// _Internal/GroupController/Interfaces/I_ContainXtsMoverGroupController
INTERFACE I_ContainXtsMoverGroupController EXTENDS I_Base

PROPERTY XtsMoverGroupController : I_XtsMoverGroupController
SET
END_SET
END_PROPERTY

END_INTERFACE

// _Internal/GroupController/Interfaces/I_XtsMoverGroupController
INTERFACE I_XtsMoverGroupController EXTENDS I_Base, I_TaskResult, I_Resettable, I_Enablable

{attribute 'monitoring' := 'call'}
PROPERTY AxesGroup : REFERENCE TO AXES_GROUP_REF
SET
END_SET
END_PROPERTY

{attribute 'monitoring':='call'}
PROPERTY GroupStatus : E_MoverGroupState
GET
END_GET
END_PROPERTY

END_INTERFACE

// _Internal/XtsSystem/Tasks/Interfaces/I_XtsMoverIdentificationTask
INTERFACE I_XtsMoverIdentificationTask EXTENDS I_XtsTask, I_Cyclic, I_XtsExecutableTask

END_INTERFACE

// _Internal/Mover/Parameters/Interfaces/I_CollisionAvoidanceGroupable
INTERFACE I_CollisionAvoidanceGroupable EXTENDS I_Base

PROPERTY AxesGroup : REFERENCE TO AXES_GROUP_REF
GET
END_GET
SET
END_SET
END_PROPERTY

{attribute 'monitoring':='call'}
PROPERTY IdentInGroup : UDINT
GET
END_GET
SET
END_SET
END_PROPERTY

END_INTERFACE

// XtsMover/XtsMover
{attribute 'no_explicit_call' := 'This FB is a CLASS and must be accessed using methods or properties'}
FUNCTION_BLOCK XtsMover EXTENDS CyclicComponent IMPLEMENTS I_XtsMover
VAR
	_Axis				  : AXIS_REF;
	_MoverTaskCollection : XtsMoverTaskCollection<15>(THIS^);
	{attribute 'hide'}
	_VirtualMover : BOOL;
	{attribute 'hide'}
	_ManualGroupControl : BOOL;
	{attribute 'hide'}
	_MoverId : UDINT;
	{attribute 'hide'}
	_Parameters	 : XtsParameterSet;
	_CurrentTask : I_XtsMoverTaskResult := NullObjects.XtsMoverTaskResult;
	_Tasks		 : _MoverTasks;
	{attribute 'hide'}
	_MoverData : I_XtsMoverData := NullObjects.XtsMoverData;
	{attribute 'hide'}
	_oldPosition : LREAL;
	{attribute 'hide'}
	_currentPosition : LREAL;
	{attribute 'hide'}
	_TrackCollection : I_XtsTrackCollection;
	{attribute 'hide'}
	_Initialized : BOOL;
	{attribute 'hide'}
	_LocalLogger : XtsLocalLogger;
	{attribute 'hide'}
	_Logger : XtsTracePublisher;

	//
	{attribute 'hide'}
	_MoverUtility : I_TcIoXtsXpuMover;
	_Positionable : PositionableBehavior(THIS^);
	{attribute 'hide'}
	_MoverStatus : XtsMoverStatus(THIS^);
END_VAR

METHOD CyclicLogic
_MoverTaskCollection.CyclicLogic();

Axis.ReadStatus();
_oldPosition := Position;
_Positionable.CyclicLogic();
END_METHOD

PROPERTY MoverTasks : I_XtsMoverTaskCollection
GET
MoverTasks := _MoverTaskCollection;
END_GET
END_PROPERTY

PROPERTY MoverUtility : I_TcIoXtsXpuMover
GET
MoverUtility := _MoverUtility;
END_GET
SET
_MoverUtility := MoverUtility;
_Positionable.MoverUtility := _MoverUtility;
END_SET
END_PROPERTY

METHOD RefreshMoverId
VAR_INPUT
	Xpu : I_TcIoXtsProcessingUnit;
END_VAR

VAR
	MoverCount : UDINT;
	i		   : UDINT;
END_VAR
IF _VirtualMover OR _MoverUtility = 0 THEN
	RETURN;
END_IF

IF Xpu = 0 THEN
	_Logger.LogMessage(Key		 := 'RefreshMoverId',
					   Value	 := 'Invalid Xpu interface provided',
					   MessageId := E_XtsLogMessage.MoverRefreshMoverIdInvalidXpu,
					   Severity	 := 3);
END_IF

FOR i := 1 TO Xpu.P_MoverCount DO
	IF _Axis.DriveAddress.TcAxisObjectId = Xpu.MoverTcIo(UDINT_TO_UINT(i)).GetAxisObjectId() THEN
		_MoverId := i;
		RETURN;
	END_IF
END_FOR

_MoverId := 0;
_Logger.LogMessage(Key		 := 'RefreshMoverId',
				   Value	 := 'AxisId not found on XPU.',
				   MessageId := E_XtsLogMessage.MoverRefreshMoverIdNoAxisObjectFound,
				   Severity	 := 1);
END_METHOD

METHOD RegisterWithParent
VAR_INPUT
	Parent	: Core.I_ContainComponents;
END_VAR
Parent.RegisterInitialize(THIS^);
SUPER^.RegisterWithParent(Parent);
END_METHOD

//Command Mover to Activate to track
METHOD ActivateTrack : I_XtsMoverTaskResult
VAR_INPUT
	TrackId : UDINT; //Track to Activate to
END_VAR

VAR
	_TrackId   : I_TakesTrackId;
	Track	   : I_XtsTrack;
END_VAR
__QUERYINTERFACE(_Tasks.ActivateTrack, _TrackId);
ActivateTrack := _Tasks.ActivateTrack;
IF _TrackId <> 0 THEN
	_TrackId.TrackId := TrackId;
END_IF

Track						  := _TrackCollection.GetById(TrackId);
_Parameters.Track			  := Track;
_CurrentTask := ActivateTrack := _Tasks.ActivateTrack.Execute();
END_METHOD

//Add Mover to CA Group
METHOD AddToGroup : I_XtsMoverTaskResult
VAR_INPUT
	Group : REFERENCE TO AXES_GROUP_REF; //Group to Add to
	Ident : UDINT; //Ident in Group
END_VAR

VAR
	LogMessage	 : TraceMessageInfo;
	LogSource	 : TraceSourceInfo;
END_VAR
AddToGroup := _Tasks.AddToGroup;
IF NOT __ISVALIDREF(Group) THEN
	LogMessage.Severity	 := 3;
	LogMessage.Message	 := 'Invalid Parameter: AxesGroup Reference on AddToGroup Command';
	LogMessage.MessageId := E_XtsLogMessage.MoverCommandErrorInvalidParameter;
	_Logger.LogMessageInstance(LogSource, LogMessage);
	RETURN;
END_IF

_Tasks.AddToGroup.AxesGroup	   REF= Group;
_Tasks.AddToGroup.IdentInGroup := Ident;
_CurrentTask := AddToGroup	   := _Tasks.AddToGroup.Execute();
END_METHOD

METHOD Disable
VAR
	LogMessage	 : TraceMessageInfo;
	LogSource	 : TraceSourceInfo;
END_VAR
_Tasks.EnableAxis.Disable();
LogSource.SourceName := _Name;
LogMessage.Severity	 := 1;
LogMessage.Message	 := 'Mover Commanded to Disable';
LogMessage.MessageId := E_XtsLogMessage.MoverCommandedToDisable;
_Logger.LogMessageInstance(LogSource, LogMessage);
END_METHOD

METHOD Enable
VAR
	LogMessage	 :TraceMessageInfo;
	LogSource	 :TraceSourceInfo;
END_VAR
_Tasks.EnableAxis.Enable();
LogSource.SourceName := _Name;
LogMessage.Severity	 := 1;
LogMessage.Message	 := 'Mover Commanded to Enable';
LogMessage.MessageId := E_XtsLogMessage.MoverCommandedToEnable;
_Logger.LogMessageInstance(LogSource, LogMessage);
END_METHOD

//Command Mover to Halt
METHOD Halt : I_XtsMoverTaskResult
VAR_INPUT
	Deceleration : LREAL; //Rate to Decelerate
	Gap			 : LREAL; //Gap to maintain to other movers
END_VAR
Halt					 := _Tasks.HaltMover;
_Parameters.Deceleration := Deceleration;
_Parameters.Gap			 := Gap;
_CurrentTask := Halt	 := _Tasks.HaltMover.Execute();
END_METHOD

//Command Mover to MoveToPosition
METHOD MoveToPosition : I_XtsMoverTaskResult
VAR_INPUT
	Position  : LREAL; //Position to move to
	Direction : Tc3_Mc3Definitions.MC_DIRECTION := Tc3_Mc3Definitions.MC_DIRECTION.mcDirectionPositive; //Direction to move
END_VAR
_Parameters.Position		   := Position;
_Parameters.Direction		   := Direction;
_CurrentTask := MoveToPosition := _Tasks.MoveToPosition.Execute();
END_METHOD

//Command Mover to Move to a Station
METHOD MoveToStation : I_XtsMoverTaskResult
VAR_INPUT
	Station : I_XtsStation; //Station to move to
END_VAR

VAR
	LogMessage	 : TraceMessageInfo;
	LogSource	 : TraceSourceInfo;
END_VAR
IF Station = 0 THEN
    LogMessage.Severity := 3;
    LogMessage.Message := 'Invalid Parameter: Station on MoveToStation Command';
    LogMessage.MessageId := E_XtsLogMessage.MoverCommandErrorInvalidParameter;
    _Logger.LogMessageInstance(LogSource, LogMessage);
    MoveToStation := NullObjects.XtsMoverTaskResult;
    RETURN;
END_IF

_Tasks.MoveToStation.Station := Station;
_CurrentTask := _Tasks.MoveToStation.Execute();
MoveToStation := _CurrentTask;
END_METHOD

//Command a Mover to Move At Velocity endlessly
METHOD MoveVelocity : I_XtsMoverTaskResult
VAR_INPUT
	Velocity  : LREAL;																					//Velocity to move at
	Direction : Tc3_Mc3Definitions.MC_DIRECTION := Tc3_Mc3Definitions.MC_DIRECTION.mcDirectionPositive; //Direction to move
END_VAR
MoveVelocity				 := _Tasks.MoveVelocity;
_Parameters.Velocity		 := Velocity;
_Parameters.Direction		 := Direction;
_CurrentTask := MoveVelocity := _Tasks.MoveVelocity.Execute();
END_METHOD

//Command Mover to remove from CA Group
METHOD RemoveFromGroup : I_XtsMoverTaskResult
VAR_INPUT
	Group : REFERENCE TO AXES_GROUP_REF; //Group to Remvoe Mover From
	Ident : UDINT;						 //Ident of Mover in Group
END_VAR

VAR
	LogMessage : TraceMessageInfo;
	LogSource  : TraceSourceInfo;
END_VAR
RemoveFromGroup := _Tasks.RemoveFromGroup;
IF NOT __ISVALIDREF(Group) THEN
	LogMessage.Severity	 := 3;
	LogMessage.Message	 := 'Invalid Parameter: AxesGroup Reference on RemoveFromGroup Command';
	LogMessage.MessageId := E_XtsLogMessage.MoverCommandErrorInvalidParameter;
	_Logger.LogMessageInstance(LogSource, LogMessage);
	RETURN;
END_IF

_Tasks.RemoveFromGroup.AxesGroup	REF= Group;
_Tasks.RemoveFromGroup.IdentInGroup := Ident;
_CurrentTask := RemoveFromGroup		:= _Tasks.RemoveFromGroup.Execute();
END_METHOD

METHOD Reset 
VAR
	LogMessage	 : TraceMessageInfo;
	LogSource	 : TraceSourceInfo;
END_VAR
_MoverTaskCollection.Reset();
_CurrentTask := _Tasks.ResetAxis.Execute();
END_METHOD

//Command Mover to Synchronize to an Axis
METHOD SyncToAxis : I_XtsMoverTaskResult
VAR_INPUT
	Master			   : REFERENCE TO AXIS_REF; //Axis to synchronize to
	MasterSyncPosition : LREAL;					//Master synchronize position			
	SlaveSyncPosition  : LREAL;					//Slave synchronize position
END_VAR

VAR
	LogMessage : TraceMessageInfo;
	LogSource  : TraceSourceInfo;
END_VAR
IF NOT __ISVALIDREF(Master) THEN
	LogMessage.Severity	 := 3;
	LogMessage.Message	 := 'Invalid Parameter: Master reference on SyncToAxis command';
	LogMessage.MessageId := E_XtsLogMessage.MoverCommandErrorInvalidParameter;
	_Logger.LogMessageInstance(LogSource, LogMessage);
	RETURN;
END_IF

_Parameters.SyncAxis.MasterAxis			REF= Master;
_Parameters.SyncAxis.MasterSyncPosition := MasterSyncPosition;
_Parameters.SyncAxis.SlaveSyncPosition	:= SlaveSyncPosition;
_CurrentTask := SyncToAxis				:= _Tasks.SyncToAxis.Execute();
END_METHOD

//Command Mover to Synchronize to another Mover
METHOD SyncToMover : I_XtsMoverTaskResult
VAR_INPUT
	Master	 : I_XtsMover; //Mover to synchronize to
	Distance : LREAL;	   //Distance between movers
END_VAR

VAR
	LogMessage : TraceMessageInfo;
	LogSource  : TraceSourceInfo;
END_VAR
IF Master = 0 THEN
	LogMessage.Severity	 := 3;
	LogMessage.Message	 := 'Invalid Parameter: Master on SyncToMover Command';
	LogMessage.MessageId := E_XtsLogMessage.MoverCommandErrorInvalidParameter;
	_Logger.LogMessageInstance(LogSource, LogMessage);
	RETURN;
END_IF

_Parameters.SyncAxis.MasterAxis			REF= Master.Axis;
_Parameters.SyncAxis.MasterSyncPosition := Master.Axis.NcToPlc.SetPos;
IF _Axis.NcToPlc.SetPos <= Master.Axis.NcToPlc.SetPos THEN
	IF Distance > 0 THEN		// ... And the Gap is Positive
		_Parameters.SyncAxis.SlaveSyncPosition		:= Master.Axis.NcToPlc.SetPos - Distance;		
	ELSE				// ... And the Gap is Negative
		_Parameters.SyncAxis.SlaveSyncPosition		:= Master.Axis.NcToPlc.SetPos - Status.CurrentTrack.Length - Distance;
	END_IF

// If the slave setpos is greater than the master...
ELSE
	IF Distance > 0 THEN		// ... And the Gap is Positive
		_Parameters.SyncAxis.SlaveSyncPosition		:= Master.Axis.NcToPlc.SetPos - Status.CurrentTrack.Length - Distance;
	ELSE				// ... And the Gap is Negative
		_Parameters.SyncAxis.SlaveSyncPosition		:= Master.Axis.NcToPlc.SetPos - Distance;		
	END_IF
END_IF
_CurrentTask := SyncToMover				:= _Tasks.SyncToAxis.Execute();
LogSource.SourceName					:= _Name;
END_METHOD

//FB_Init is always available implicitly and it is used primarily for initialization.

//The return value is not evaluated. For a specific influence, you can also declare the

//methods explicitly and provide additional code there with the standard initialization

//code. You can evaluate the return value.
METHOD FB_Init : BOOL
VAR_INPUT
	bInitRetains : BOOL; // TRUE: the retain variables are initialized (reset warm / reset cold)
	bInCopyCode	 : BOOL; // TRUE: the instance will be copied to the copy code afterward (online change)
	Name		 : T_MaxString;
	MoverData	 : I_XtsMoverData;		   //Optional MoverData assignment
	System		 : I_ContainXtsMovers; //Optional Self Registration with an Xts System
END_VAR
_MoverTaskCollection.AddTask(_Tasks.EnableAxis);
_MoverTaskCollection.AddTask(_Tasks.ResetAxis);
_MoverTaskCollection.AddTask(_Tasks.MoveToPosition);
_MoverTaskCollection.AddTask(_Tasks.MoveToStation);
_MoverTaskCollection.AddTask(_Tasks.MoveVelocity);
_MoverTaskCollection.AddTask(_Tasks.HaltMover);
_MoverTaskCollection.AddTask(_Tasks.AddToGroup);
_MoverTaskCollection.AddTask(_Tasks.RemoveFromGroup);
_MoverTaskCollection.AddTask(_Tasks.ActivateTrack);
_MoverTaskCollection.AddTask(_Tasks.SyncToAxis);
_Logger.Subscribe(_LocalLogger);
IF XtsCoreParameters.TcEventLoggerEnabled THEN
	_Logger.Subscribe(XtsTrace.EventLogger);
END_IF

IF MoverData <> 0 THEN
	_MoverData := MoverData;
END_IF

IF System <> 0 THEN
	System.Movers.AddItem(THIS^);
	RegisterWithParent(System);
END_IF
END_METHOD

METHOD Initialize
VAR
	CurrentTrackOtcid : OTCID;
END_VAR
IF _TrackCollection = 0 THEN
	RETURN;
END_IF


IF _MoverUtility = 0 OR _VirtualMover THEN
	_Initialized := TRUE;	
	RETURN;
END_IF

CurrentTrackOtcid := _MoverUtility.GetActiveTrackObjectId();
_TrackCollection.ResetIterator();
WHILE _TrackCollection.MoveToNext DO
	IF _TrackCollection.Current.Otcid = CurrentTrackOtcid THEN
		_MoverStatus.CurrentTrack := _TrackCollection.Current;
		EXIT;
	END_IF
END_WHILE

_Initialized := TRUE;
END_METHOD

{attribute 'monitoring' := 'call'}
PROPERTY Initialized : BOOL
GET
Initialized := _Initialized;
END_GET
SET
_Initialized := Initialized;
END_SET
END_PROPERTY

PROPERTY Axis : REFERENCE TO Tc2_MC2.AXIS_REF
GET
Axis REF= _Axis;
END_GET
END_PROPERTY

{attribute 'monitoring' := 'call'}
PROPERTY InhibitFeedBackward : BOOL
GET
InhibitFeedBackward := _Tasks.EnableAxis.InhibitFeedBackward;
END_GET
SET
_Tasks.EnableAxis.InhibitFeedBackward := InhibitFeedBackward;
END_SET
END_PROPERTY

{attribute 'monitoring' := 'call'}
PROPERTY InhibitFeedForward : BOOL
GET
InhibitFeedForward := _Tasks.EnableAxis.InhibitFeedForward;
END_GET
SET
_Tasks.EnableAxis.InhibitFeedForward := InhibitFeedForward;
END_SET
END_PROPERTY

{attribute 'monitoring':='call'}
PROPERTY InPosition : BOOL
GET
VAR
	difference : LREAL;
END_VAR
difference := ABS(Position - _Parameters.Position);
InPosition := MIN(difference, _Parameters.Track.Length - difference) < 1.0 AND (NOT _Tasks.MoveToPosition.Busy OR NOT _Tasks.MoveToStation.Busy);
END_GET
END_PROPERTY

{attribute 'monitoring':='call'}
PROPERTY InVelocity : BOOL
GET
InVelocity := ABS(_Axis.NcToPlc.ActVelo -  _Axis.NcToPlc.SetVelo) < 10.0 AND _Axis.NcToPlc.SetVelo <> 0;
END_GET
END_PROPERTY

PROPERTY LastCyclePosition : LREAL
GET
LastCyclePosition := _oldPosition;
END_GET
END_PROPERTY

{attribute 'monitoring':='call'}
PROPERTY ManualGroupControl : BOOL
GET
ManualGroupControl := _ManualGroupControl;
END_GET
SET
_ManualGroupControl := ManualGroupControl;
END_SET
END_PROPERTY

{attribute 'monitoring':='call'}
PROPERTY MoverData : I_XtsMoverData
GET
MoverData := _MoverData;
END_GET
SET
_MoverData := MoverData;
END_SET
END_PROPERTY

{attribute 'monitoring':='call'}
PROPERTY MoverId : UDINT
GET
MoverId := _MoverId;
END_GET
END_PROPERTY

{attribute 'monitoring' := 'call'}
PROPERTY Override : LREAL
SET
_Tasks.EnableAxis.Override := Override;
END_SET
END_PROPERTY

{attribute 'monitoring':='call'}
PROPERTY Parameters : I_XtsParameterSet
GET
Parameters := _Parameters;
END_GET
SET
END_SET
END_PROPERTY

{attribute 'monitoring':='call'}
PROPERTY Position : LREAL
GET
VAR
	tmp : LREAL;
END_VAR
Position := _Positionable.Position;
END_GET
END_PROPERTY

{attribute 'hide'}
PROPERTY Tracks : I_XtsTrackCollection
GET
Tracks := _TrackCollection;
END_GET
SET
_TrackCollection := Tracks;
//Reset the Activate Task axis assignment to refresh track collection assignment
_Tasks.ActivateTrack.Axis := THIS^;
END_SET
END_PROPERTY

{attribute 'monitoring':='call'}
PROPERTY VirtualMover : BOOL
GET
VirtualMover := _VirtualMover;
END_GET
SET
_VirtualMover := VirtualMover;
END_SET
END_PROPERTY

{attribute 'monitoring':='call'}
PROPERTY Busy : BOOL
GET
Busy := _MoverTaskCollection.Busy;
END_GET
END_PROPERTY

{attribute 'monitoring':='call'}
//Last Commanded Task to Mover
PROPERTY CurrentTask : I_XtsMoverTaskResult
GET
CurrentTask := _CurrentTask;
END_GET
END_PROPERTY

{attribute 'monitoring' := 'call'}
PROPERTY Enabled : BOOL
GET
Enabled := _Tasks.EnableAxis.Enabled;
END_GET
END_PROPERTY

{attribute 'monitoring':='call'}
PROPERTY Error : BOOL
GET
Error := _MoverTaskCollection.Error;
END_GET
END_PROPERTY

{attribute 'monitoring':='call'}
PROPERTY ErrorId : UDINT
GET
IF _Axis.Status.ErrorID <> 0 THEN
	ErrorId := _Axis.Status.ErrorID;
	RETURN;
END_IF

ErrorId := _MoverTaskCollection.ErrorId;
END_GET
END_PROPERTY

{attribute 'monitoring':='call'}
PROPERTY Status : I_XtsMoverStatus
GET
Status := _MoverStatus;
END_GET
END_PROPERTY

{attribute 'monitoring':='call'}
PROPERTY CommandLog : I_XtsLocalLog
GET
CommandLog := _LocalLogger;
END_GET
END_PROPERTY

PROPERTY TracePublisher : I_XtsTracePublisher
GET
TracePublisher := _Logger;
END_GET
END_PROPERTY

METHOD AcceptMoverVisitor
VAR_INPUT
	MoverVisitor : I_XtsMoverVisitor;
END_VAR
MoverVisitor.VisitMover(THIS^);
END_METHOD

END_FUNCTION_BLOCK

// _Internal/Mover/MoverTaskBase/XtsMoverTaskCollection
{attribute 'no_explicit_call' := 'This FB is a CLASS and must be accessed using methods or properties'}
FUNCTION_BLOCK XtsMoverTaskCollection
VAR_GENERIC CONSTANT
	MaxCount : UDINT := 10;
END_VAR IMPLEMENTS I_XtsMoverTaskCollection, I_Cyclic
VAR
	MotionTasks : ARRAY[0..MaxCount - 1] OF I_XtsMoverTask;
	_TaskCount	: UDINT;
	Axis		: I_AxisRef;
	_ErrorId	: UDINT;
	_Busy		: BOOL;
	_Error		: BOOL;
	_ErrorTask	: T_MaxString;
	{attribute 'hide'}
	_Logger : I_XtsLogger;
	{attribute 'hide'}
	LogSource : TraceSourceInfo;
	{attribute 'hide'}
	LogMessage : TraceMessageInfo;
END_VAR

PROPERTY Busy : BOOL
GET
Busy := _Busy;
END_GET
END_PROPERTY

PROPERTY Error : BOOL
GET
Error := _Error;
END_GET
END_PROPERTY

PROPERTY ErrorId : UDINT
GET
ErrorId := _ErrorId;
END_GET
END_PROPERTY

PROPERTY ErrorTask : T_MaxString
GET
ErrorTask := _ErrorTask;
END_GET
END_PROPERTY

METHOD AddTask : BOOL
VAR_INPUT
	Task	: I_XtsMoverTask;
END_VAR
IF _TaskCount = MaxCount THEN
	AddTask := FALSE;
	RETURN;
END_IF
Task.Axis := Axis;
MotionTasks[Task.TaskId] := Task;
_TaskCount := _TaskCount + 1;
AddTask := TRUE;
END_METHOD

METHOD CyclicLogic
VAR
	i	 : UDINT;
END_VAR
_Busy := FALSE;
FOR i := 0 TO MaxCount - 1 DO
	IF MotionTasks[i] = 0 THEN
		CONTINUE;
	END_IF

	MotionTasks[i].CyclicLogic();
	IF MotionTasks[i].Busy THEN
		_Busy := TRUE;
	END_IF

	IF MotionTasks[i].Error AND NOT _Error THEN
		LogMessage.Message	 := CONCAT('Mover Task: ', CONCAT(MotionTasks[i].TaskName, CONCAT(' ErrorId: ', TO_STRING(MotionTasks[i].ErrorId))));
		LogMessage.MessageId := E_XtsLogMessage.MoverCommandGeneralTaskError;
		LogMessage.Severity	 := 3;
		_Logger.LogMessageInstance(LogSource, LogMessage);
		_Error	   := TRUE;
		_ErrorId   := MotionTasks[i].ErrorId;
		_ErrorTask := MotionTasks[i].TaskName;
	END_IF
END_FOR
END_METHOD

//FB_Init is always available implicitly and it is used primarily for initialization.

//The return value is not evaluated. For a specific influence, you can also declare the

//methods explicitly and provide additional code there with the standard initialization

//code. You can evaluate the return value.
METHOD FB_Init : BOOL
VAR_INPUT
	bInitRetains : BOOL; // TRUE: the retain variables are initialized (reset warm / reset cold)
	bInCopyCode	 : BOOL; // TRUE: the instance will be copied to the copy code afterward (online change)
	Axis		 : I_AxisRef;
END_VAR
VAR
	Mover : I_XtsMover;
END_VAR
THIS^.Axis			 := Axis;
LogSource.SourceName := 'Task Collection';
__QUERYINTERFACE(Axis, Mover);
__QUERYINTERFACE(Mover.TracePublisher, _Logger);
END_METHOD

METHOD GetTaskById : I_XtsMoverTask
VAR_INPUT
	TaskId : MoverTaskID;
END_VAR
GetTaskById := MotionTasks[TaskId];
END_METHOD

METHOD GetTaskByName : I_XtsMoverTask
VAR_INPUT
	Name : T_MaxString;
END_VAR

VAR
	i	 : UDINT;
END_VAR
GetTaskByName := NullObjects.XtsMoverTask;
FOR i:=0 TO _TaskCount - 1 DO
	IF MotionTasks[i].TaskName = Name THEN
		GetTaskByName := MotionTasks[i];
		RETURN;
	END_IF
END_FOR
END_METHOD

METHOD RemoveTaskById : BOOL
VAR_INPUT
	TaskId : MoverTaskId;
END_VAR
IF MotionTasks[TaskId] = 0 THEN
	RETURN;
END_IF

MotionTasks[TaskId] := 0;
_TaskCount			:= _TaskCount - 1;
RemoveTaskById		:= TRUE;
END_METHOD

METHOD RemoveTaskByInstance : BOOL
VAR_INPUT
	Task : I_XtsMoverTask;
END_VAR
IF MotionTasks[Task.TaskId] = 0 THEN
	RETURN;
END_IF

MotionTasks[Task.TaskId] := 0;
_TaskCount				 := _TaskCount - 1;
RemoveTaskByInstance	 := TRUE;
END_METHOD

METHOD Reset
VAR_INPUT
END_VAR
VAR
	i : UDINT;
END_VAR
_Error	   := FALSE;
_ErrorId   := 0;
_ErrorTask := '';
FOR i := 0 TO MaxCount - 1 DO
	IF MotionTasks[i] = 0 THEN
		CONTINUE;
	END_IF
	MotionTasks[i].Reset();
END_FOR
END_METHOD

END_FUNCTION_BLOCK

// _Internal/Mover/Tasks/_MoverTasks
{attribute 'no_explicit_call' := 'This FB is a CLASS and must be accessed using methods or properties'}
FUNCTION_BLOCK _MoverTasks
VAR
	_DefaultTask	 : _DefaultMoverTasks;
	_MoveToPosition	 : I_XtsMoverTask		:= _DefaultTask.MoveToPositionCA;
	_MoveVelocity	 : I_XtsMoverTask		:= _DefaultTask.MoveVelocity;
	_HaltMoverCA	 : I_XtsMoverTask		:= _DefaultTask.HaltMoverCA;
	_AddToGroup		 : I_AxesGroupTask		:= _DefaultTask.AddToGroup;
	_RemoveFromGroup : I_AxesGroupTask		:= _DefaultTask.RemoveFromGroup;
	_MoveToStation	 : I_MoveToStationTask	:= _DefaultTask.MoveToStation;
	_ActivateTrack	 : I_XtsMoverTask		:= _DefaultTask.ActivateTrack;
	_EnableAxis		 : I_EnableXtsMoverTask := _DefaultTask.EnableAxis;
	_ResetAxis		 : I_XtsMoverTask		:= _DefaultTask.ResetAxis;
	_SyncToAxis		 : I_XtsMoverTask		:= _DefaultTask.SyncToAxis;
END_VAR

PROPERTY ActivateTrack : I_XtsMoverTask
GET
ActivateTrack := _ActivateTrack;
END_GET
SET
_ActivateTrack := ActivateTrack;
END_SET
END_PROPERTY

PROPERTY AddToGroup : I_AxesGroupTask
GET
AddToGroup := _AddToGroup;
END_GET
SET
_AddToGroup := AddToGroup;
END_SET
END_PROPERTY

PROPERTY EnableAxis : I_EnableXtsMoverTask
GET
EnableAxis := _EnableAxis;
END_GET
SET
_EnableAxis := EnableAxis;
END_SET
END_PROPERTY

PROPERTY HaltMover : I_XtsMoverTask
GET
HaltMover := _HaltMoverCA;
END_GET
SET
_HaltMoverCA := HaltMover;
END_SET
END_PROPERTY

PROPERTY MoveToPosition : I_XtsMoverTask
GET
MoveToPosition := _MoveToPosition;
END_GET
SET
_MoveToPosition := MoveToPosition;
END_SET
END_PROPERTY

PROPERTY MoveToStation : I_MoveToStationTask
GET
MoveToStation := _MoveToStation;
END_GET
SET
_MoveToStation := MoveToStation;
END_SET
END_PROPERTY

PROPERTY MoveVelocity : I_XtsMoverTask
GET
MoveVelocity := _MoveVelocity;
END_GET
SET
_MoveVelocity := MoveVelocity;
END_SET
END_PROPERTY

PROPERTY RemoveFromGroup : I_AxesGroupTask
GET
RemoveFromGroup := _RemoveFromGroup;
END_GET
SET
_RemoveFromGroup := RemoveFromGroup;
END_SET
END_PROPERTY

PROPERTY ResetAxis : I_XtsMoverTask
GET
ResetAxis := _ResetAxis;
END_GET
SET
_ResetAxis := ResetAxis;
END_SET
END_PROPERTY

METHOD ResetToDefault
VAR_INPUT
END_VAR
_MoveToPosition	 := _DefaultTask.MoveToPositionCA;
_MoveVelocity	 := _DefaultTask.MoveVelocity;
_HaltMoverCA	 := _DefaultTask.HaltMoverCA;
_AddToGroup		 := _DefaultTask.AddToGroup;
_RemoveFromGroup := _DefaultTask.RemoveFromGroup;
_MoveToStation	 := _DefaultTask.MoveToStation;
_ActivateTrack	 := _DefaultTask.ActivateTrack;
_EnableAxis		 := _DefaultTask.EnableAxis;
_ResetAxis		 := _DefaultTask.ResetAxis;
_SyncToAxis		 := _DefaultTask.SyncToAxis;
END_METHOD

PROPERTY SyncToAxis : I_XtsMoverTask
GET
SyncToAxis := _SyncToAxis;
END_GET
SET
_SyncToAxis := SyncToAxis;
END_SET
END_PROPERTY

END_FUNCTION_BLOCK

// _Internal/Mover/Tasks/_DefaultMoverTasks
{attribute 'no_explicit_call' := 'This FB is a CLASS and must be accessed using methods or properties'}
FUNCTION_BLOCK _DefaultMoverTasks
VAR
	NullMotionTask	 : NullXtsMoverTask;
	EnableAxis		 : EnableAxisTask;
	AddToGroup		 : AddToGroupTask;
	RemoveFromGroup	 : RemoveFromGroupTask;
	HaltMoverCA		 : HaltMoverCATask;
	MoveToPositionCA : MoveToPositionCATask;
	MoveVelocity	 : MoveVelocityTask;
	MoveToStation	 : MoveToStationTask;
	ActivateTrack	 : ActivateTrackTask;
	ResetAxis		 : ResetAxisTask;
	SyncToAxis		 : SyncToAxisTask;
END_VAR

END_FUNCTION_BLOCK

// _Internal/NullObjects/NullXtsMoverTask
{attribute 'no_explicit_call' := 'This FB is a CLASS and must be accessed using methods or properties'}
{attribute 'conditionalshow'}
{warning disable C0094}
{warning disable C0568}
FUNCTION_BLOCK NullXtsMoverTask EXTENDS XtsMoverTaskResult IMPLEMENTS I_XtsMoverTask, I_NullObject
VAR
END_VAR

PROPERTY Axis : I_AxisRef
GET
END_GET
SET
END_SET
END_PROPERTY

METHOD CyclicLogic
END_METHOD

METHOD Execute : I_XtsMoverTaskResult
Execute := NullObjects.XtsMoverTaskResult;
END_METHOD

METHOD Reset
END_METHOD

PROPERTY TaskId : MoverTaskId
GET
END_GET
END_PROPERTY

{attribute 'monitoring':='call'}
PROPERTY TaskName : STRING
GET
TaskName := 'No task active';
END_GET
END_PROPERTY

END_FUNCTION_BLOCK

// _Internal/Mover/Tasks/EnableAxisTask
{attribute 'no_explicit_call' := 'This FB is a CLASS and must be accessed using methods or properties'}
FUNCTION_BLOCK EnableAxisTask EXTENDS XtsMoverTaskResult IMPLEMENTS I_EnableXtsMoverTask
VAR
	_Axis			   : I_AxisRef;
	_DefaultAxisEnable : PowerAxis;
	EnableAxisFb	   : I_Power := _DefaultAxisEnable;
	{attribute 'hide'}
	_InhibitFeedForward : BOOL;
	{attribute 'hide'}
	_InhibitFeedBackward : BOOL;
END_VAR

PROPERTY Axis : I_AxisRef
GET
Axis := _Axis;
END_GET
SET
_Axis := Axis;
END_SET
END_PROPERTY

METHOD CyclicLogic
EnableAxisFb.Enable_Positive := NOT _InhibitFeedForward;
EnableAxisFb.Enable_Negative := NOT _InhibitFeedBackward;
_DefaultAxisEnable(Axis := _Axis.Axis);
_Error	 := EnableAxisFb.Error;
_Busy	 := EnableAxisFb.Busy AND NOT EnableAxisFb.Status;
_ErrorId := EnableAxisFb.ErrorId;
END_METHOD

METHOD Disable
EnableAxisFb.Enable := FALSE;
END_METHOD

{attribute 'monitoring' := 'call'}
PROPERTY Disabled : BOOL
GET
Disabled := EnableAxisFb.Status = FALSE;
END_GET
END_PROPERTY

METHOD Enable
EnableAxisFb.Enable := TRUE;
END_METHOD

{attribute 'monitoring' := 'call'}
PROPERTY Enabled : BOOL
GET
Enabled := EnableAxisFb.Status;
END_GET
END_PROPERTY

METHOD Execute : I_XtsMoverTaskResult
Execute := THIS^;
END_METHOD

//FB_Init is always available implicitly and it is used primarily for initialization.

//The return value is not evaluated. For a specific influence, you can also declare the

//methods explicitly and provide additional code there with the standard initialization

//code. You can evaluate the return value.
METHOD FB_Init : BOOL
VAR_INPUT
	bInitRetains : BOOL; // TRUE: the retain variables are initialized (reset warm / reset cold)
	bInCopyCode	 : BOOL; // TRUE: the instance will be copied to the copy code afterward (online change)
END_VAR
_TaskName := 'Enable Axis';
_TaskId	  := MoverTaskId.ENABLE;
END_METHOD

{attribute 'monitoring' := 'call'}
PROPERTY InhibitFeedBackward : BOOL
GET
InhibitFeedBackward := _InhibitFeedBackward;
END_GET
SET
_InhibitFeedBackward := InhibitFeedBackward;
END_SET
END_PROPERTY

{attribute 'monitoring' := 'call'}
PROPERTY InhibitFeedForward : BOOL
GET
InhibitFeedForward := _InhibitFeedForward;
END_GET
SET
_InhibitFeedForward := InhibitFeedForward;
END_SET
END_PROPERTY

{attribute 'monitoring' := 'call'}
PROPERTY Override : LREAL
SET
EnableAxisFb.Override := Override;
END_SET
END_PROPERTY

METHOD Reset
_Error				 := FALSE;
_ErrorID			 := 0;
_Busy				 := FALSE;
ExecuteWatchdog		 := 0;
_CommandExecuted	 := FALSE;
END_METHOD

END_FUNCTION_BLOCK

// _Internal/Mover/Tasks/Interfaces/I_EnableXtsMoverTask
INTERFACE I_EnableXtsMoverTask EXTENDS I_XtsMoverTask, I_Cyclic

METHOD Disable
END_METHOD

{attribute 'monitoring' := 'call'}
PROPERTY Disabled : BOOL
GET
END_GET
END_PROPERTY

METHOD Enable
END_METHOD

{attribute 'monitoring' := 'call'}
PROPERTY Enabled : BOOL
GET
END_GET
END_PROPERTY

{attribute 'monitoring' := 'call'}
PROPERTY InhibitFeedBackward : BOOL
GET
END_GET
SET
END_SET
END_PROPERTY

{attribute 'monitoring' := 'call'}
PROPERTY InhibitFeedForward : BOOL
GET
END_GET
SET
END_SET
END_PROPERTY

{attribute 'monitoring' := 'call'}
PROPERTY Override : LREAL
SET
END_SET
END_PROPERTY

END_INTERFACE

// _Internal/Mover/Tasks/Wrappers/PowerAxis
FUNCTION_BLOCK PowerAxis IMPLEMENTS I_Power
VAR
	_mcPower : MC_Power;
END_VAR

VAR_IN_OUT
	Axis : Tc2_Mc2.AXIS_REF;
END_VAR

_mcPower(Axis := Axis);

{attribute 'monitoring':='call'}
PROPERTY BufferMode : MC_BufferMode
GET
BufferMode := _mcPower.BufferMode;
END_GET
SET
_mcPower.BufferMode := BufferMode;
END_SET
END_PROPERTY

{attribute 'monitoring':='call'}
PROPERTY Enable : BOOL
GET
Enable := _mcPower.Enable;
END_GET
SET
_mcPower.Enable := Enable;
END_SET
END_PROPERTY

{attribute 'monitoring':='call'}
PROPERTY Enable_Negative : BOOL;
GET
Enable_Negative := _mcPower.Enable_Negative;
END_GET
SET
_mcPower.Enable_Negative := Enable_Negative;
END_SET
END_PROPERTY

{attribute 'monitoring':='call'}
PROPERTY Enable_Positive : BOOL
GET
Enable_Positive := _mcPower.Enable_Positive;
END_GET
SET
_mcPower.Enable_Positive := Enable_Positive;
END_SET
END_PROPERTY

PROPERTY Options : ST_PowerOptions
GET
Options := _mcPower.Options;
END_GET
SET
_mcPower.Options := Options;
END_SET
END_PROPERTY

{attribute 'monitoring':='call'}
PROPERTY Override : MC_LREAL
GET
Override := _mcPower.Override;
END_GET
SET
_mcPower.Override := Override;
END_SET
END_PROPERTY

{attribute 'monitoring':='call'}
PROPERTY Busy : BOOL
GET
Busy := _mcPower.Busy;
END_GET
END_PROPERTY

{attribute 'monitoring':='call'}
PROPERTY Error : BOOL
GET
Error := _mcPower.Error;
END_GET
END_PROPERTY

{attribute 'monitoring':='call'}
PROPERTY ErrorId : UDINT
GET
ErrorId := _mcPower.ErrorID;
END_GET
END_PROPERTY

{attribute 'monitoring':='call'}
PROPERTY Status : BOOL
GET
Status := _mcPower.Status;
END_GET
END_PROPERTY

END_FUNCTION_BLOCK

// _Internal/Mover/Tasks/Wrappers/Interfaces/I_Power
INTERFACE I_Power EXTENDS I_Base

{attribute 'monitoring':='call'}
PROPERTY BufferMode : MC_BufferMode
GET
END_GET
SET
END_SET
END_PROPERTY

{attribute 'monitoring':='call'}
PROPERTY Enable : BOOL
GET
END_GET
SET
END_SET
END_PROPERTY

{attribute 'monitoring':='call'}
PROPERTY Enable_Negative : BOOL;
GET
END_GET
SET
END_SET
END_PROPERTY

{attribute 'monitoring':='call'}
PROPERTY Enable_Positive : BOOL
GET
END_GET
SET
END_SET
END_PROPERTY

PROPERTY Options : ST_PowerOptions
GET
END_GET
SET
END_SET
END_PROPERTY

{attribute 'monitoring':='call'}
PROPERTY Override : MC_LREAL
GET
END_GET
SET
END_SET
END_PROPERTY

{attribute 'monitoring':='call'}
PROPERTY Busy : BOOL
GET
END_GET
END_PROPERTY

{attribute 'monitoring':='call'}
PROPERTY Error : BOOL
GET
END_GET
END_PROPERTY

{attribute 'monitoring':='call'}
PROPERTY ErrorId : UDINT
GET
END_GET
END_PROPERTY

{attribute 'monitoring':='call'}
PROPERTY Status : BOOL
GET
END_GET
END_PROPERTY

END_INTERFACE

// _Internal/Mover/Tasks/AddToGroupTask
{attribute 'no_explicit_call' := 'This FB is a CLASS and must be accessed using methods or properties'}
FUNCTION_BLOCK AddToGroupTask EXTENDS XtsMoverTaskResult IMPLEMENTS I_AxesGroupTask
VAR
	_Axis				   : I_AxisRef;
	_MoverStatus		   : I_XtsMoverStatus;
	_DefaultAddAxisToGroup : AddAxisToGroup;
	AddToGroupFb		   : I_AxisOnGroup := _DefaultAddAxisToGroup;
	_AxesGroup			   : REFERENCE TO AXES_GROUP_REF;
	_Ident				   : UDINT;
	Executed			   : BOOL;
END_VAR

PROPERTY AxesGroup : REFERENCE TO AXES_GROUP_REF
GET
AxesGroup REF= _AxesGroup;
END_GET
SET
_AxesGroup REF= AxesGroup;
END_SET
END_PROPERTY

PROPERTY Axis : I_AxisRef
GET
Axis := _Axis;
END_GET
SET
VAR
	Mover : I_XtsMover;
END_VAR
_Axis := Axis;
__QUERYINTERFACE(_Axis, Mover);
__QUERYINTERFACE(Mover.TracePublisher, _Logger);
_MoverStatus := Mover.Status;
END_SET
END_PROPERTY

METHOD CyclicLogic
SUPER^.CyclicLogic(); //Watchdog handling
_DefaultAddAxisToGroup(Axis := _Axis.Axis, AxesGroup := _AxesGroup);
AddToGroupFb.Execute := FALSE;
_Busy				 := AddToGroupFb.Busy;
IF _Busy THEN
	RETURN;
END_IF

(*Latch signals if they are set by the FB instance itself.
Only reset them in the event of an Task.Execute() call*)
IF Executed THEN
	Executed				  := FALSE;
	_MoverStatus.IdentInGroup := _Ident;
END_IF

_Error := AddToGroupFb.Error OR _Error;
IF AddToGroupFb.ErrorId <> 0 THEN
	_ErrorId := AddToGroupFb.ErrorId;
END_IF
END_METHOD

METHOD Execute : I_XtsMoverTaskResult
Execute			:= THIS^;
ExecuteWatchdog := ExecuteWatchdog + 1;
IF NOT __ISVALIDREF(_AxesGroup) OR _Ident = 0 THEN
	//TODO: error message
	RETURN;
END_IF

IF _Busy OR _CommandExecuted THEN
	RETURN;
END_IF

_Error					  := FALSE;
_ErrorId				  := 0;
_Busy					  := TRUE;
AddToGroupFb.IdentInGroup := _Ident;
AddToGroupFb.Execute	  := TRUE;
_CommandExecuted		  := TRUE;
Executed				  := TRUE;
LogMessage.Severity		  := 1;
LogMessage.Message		  := 'Commanded to Add to Group.';
LogMessage.MessageId	  := E_XtsLogMessage.MoverCommandedToAddToGroup;
_Logger.LogMessageInstance(LogSource, LogMessage);
END_METHOD

//FB_Init is always available implicitly and it is used primarily for initialization.

//The return value is not evaluated. For a specific influence, you can also declare the

//methods explicitly and provide additional code there with the standard initialization

//code. You can evaluate the return value.
METHOD FB_Init : BOOL
VAR_INPUT
	bInitRetains : BOOL; // TRUE: the retain variables are initialized (reset warm / reset cold)
	bInCopyCode	 : BOOL; // TRUE: the instance will be copied to the copy code afterward (online change)
END_VAR
_TaskName			 := 'Add Axis To Group';
_TaskId				 := MoverTaskId.ADD_TO_GROUP;
LogSource.SourceName := _TaskName;
LogSource.SourceId	 := _TaskId;
END_METHOD

{attribute 'monitoring':='call'}
PROPERTY IdentInGroup : UDINT
GET
IdentInGroup := _Ident;
END_GET
SET
_Ident := IdentInGroup;
END_SET
END_PROPERTY

METHOD Reset
Executed			 := FALSE;
_Error				 := FALSE;
_ErrorID			 := 0;
_Busy				 := FALSE;
ExecuteWatchdog		 := 0;
_CommandExecuted	 := FALSE;
AddToGroupFb.Execute := FALSE;
END_METHOD

END_FUNCTION_BLOCK

// _Internal/Mover/Tasks/Interfaces/I_AxesGroupTask
INTERFACE I_AxesGroupTask EXTENDS I_Base, I_XtsMoverTask, I_CollisionAvoidanceGroupable

END_INTERFACE

// _Internal/Mover/Tasks/Wrappers/AddAxisToGroup
FUNCTION_BLOCK AddAxisToGroup IMPLEMENTS I_AxisOnGroup
VAR
	_AddAxisToGroup : MC_AddAxisToGroup;
	_Ident			: UDINT;
END_VAR

VAR_IN_OUT
	Axis	  : Tc2_Mc2.AXIS_REF;
	AxesGroup : Tc3_McCoordinatedMotion.AXES_GROUP_REF;
END_VAR

_AddAxisToGroup(Axis := Axis, AxesGroup := AxesGroup);

{attribute 'monitoring':='call'}
PROPERTY Execute : BOOL
GET
Execute := _AddAxisToGroup.Execute;
END_GET
SET
_AddAxisToGroup.Execute := Execute;
END_SET
END_PROPERTY

{attribute 'monitoring':='call'}
PROPERTY IdentInGroup : UDINT
GET
IdentInGroup := _Ident;
END_GET
SET
_Ident := IdentInGroup;
_AddAxisToGroup.IdentInGroup :=UDINT_TO_IDENTINGROUP(IdentInGroup);
END_SET
END_PROPERTY

{attribute 'monitoring':='call'}
PROPERTY Busy : BOOL
GET
Busy := _AddAxisToGroup.Busy;
END_GET
END_PROPERTY

{attribute 'monitoring':='call'}
PROPERTY Done : BOOL
GET
Done := _AddAxisToGroup.Done;
END_GET
END_PROPERTY

{attribute 'monitoring':='call'}
PROPERTY Error : BOOL
GET
Error := _AddAxisToGroup.Error;
END_GET
END_PROPERTY

{attribute 'monitoring':='call'}
PROPERTY ErrorId : UDINT
GET
ErrorId := _AddAxisToGroup.ErrorId;
END_GET
END_PROPERTY

END_FUNCTION_BLOCK

// _Internal/Mover/Tasks/Wrappers/Interfaces/I_AxisOnGroup
INTERFACE I_AxisOnGroup EXTENDS I_Base

{attribute 'monitoring':='call'}
PROPERTY Execute : BOOL
GET
END_GET
SET
END_SET
END_PROPERTY

{attribute 'monitoring':='call'}
PROPERTY IdentInGroup : UDINT
GET
END_GET
SET
END_SET
END_PROPERTY

{attribute 'monitoring':='call'}
PROPERTY Busy : BOOL
GET
END_GET
END_PROPERTY

{attribute 'monitoring':='call'}
PROPERTY Error : BOOL
GET
END_GET
END_PROPERTY

{attribute 'monitoring':='call'}
PROPERTY ErrorId : UDINT
GET
END_GET
END_PROPERTY

END_INTERFACE

// _Internal/Mover/Tasks/RemoveFromGroupTask
{attribute 'no_explicit_call' := 'This FB is a CLASS and must be accessed using methods or properties'}
FUNCTION_BLOCK RemoveFromGroupTask EXTENDS XtsMoverTaskResult IMPLEMENTS I_AxesGroupTask
VAR
	_Axis						: I_AxisRef;
	_MoverStatus				: I_XtsMoverStatus;
	_DefaultRemoveAxisFromGroup : RemoveAxisFromGroup;
	RemoveFromGroupFb			: I_AxisOnGroup := _DefaultRemoveAxisFromGroup;
	_AxesGroup					: REFERENCE TO AXES_GROUP_REF;
	_Ident						: UDINT;
	Executed					: BOOL;
END_VAR

PROPERTY AxesGroup : REFERENCE TO AXES_GROUP_REF
GET
AxesGroup REF= _AxesGroup;
END_GET
SET
_AxesGroup REF= AxesGroup;
END_SET
END_PROPERTY

PROPERTY Axis : I_AxisRef
GET
Axis := _Axis;
END_GET
SET
VAR
	Mover : I_XtsMover;
END_VAR
_Axis := Axis;
__QUERYINTERFACE(_Axis, Mover);
__QUERYINTERFACE(Mover.TracePublisher, _Logger);
_MoverStatus := Mover.Status;
END_SET
END_PROPERTY

METHOD CyclicLogic
SUPER^.CyclicLogic(); //Watchdog handling
_DefaultRemoveAxisFromGroup(AxesGroup := _AxesGroup);
RemoveFromGroupFb.Execute := FALSE;
_Busy					  := RemoveFromGroupFb.Busy;
IF _Busy THEN
	RETURN;
END_IF

(*Latch signals if they are set by the FB instance itself.
Only reset them in the event of an Task.Execute() call*)
IF Executed AND _MoverStatus.IdentInGroup <> 0 THEN
	Executed				  := FALSE;
	_MoverStatus.IdentInGroup := 0;
END_IF

_Error := RemoveFromGroupFb.Error OR _Error;
IF RemoveFromGroupFb.ErrorId <> 0 THEN
	_ErrorId := RemoveFromGroupFb.ErrorId;
END_IF
END_METHOD

METHOD Execute : I_XtsMoverTaskResult
Execute			:= THIS^;
ExecuteWatchdog := ExecuteWatchdog + 1;
IF NOT __ISVALIDREF(_AxesGroup) THEN
	//TODO: error message
	RETURN;
END_IF

IF _Busy OR _CommandExecuted THEN
	RETURN;
END_IF

LogMessage.Severity	 := 1;
LogMessage.Message	 := 'Commanded to Remove From Group';
LogMessage.MessageId := E_XtsLogMessage.MoverCommandedToRemoveFromGroup;
_Logger.LogMessageInstance(LogSource, LogMessage);
IF NOT _MoverStatus.MoverInGroup THEN
	_Error	 := FALSE;
	_ErrorId := 0;
	_Busy	 := FALSE;
	RETURN;
END_IF

_Error						   := FALSE;
_ErrorId					   := 0;
_Busy						   := TRUE;
RemoveFromGroupFb.IdentInGroup := _Ident;
RemoveFromGroupFb.Execute	   := TRUE;
Executed					   := TRUE;
_CommandExecuted			   := TRUE;
END_METHOD

//FB_Init is always available implicitly and it is used primarily for initialization.

//The return value is not evaluated. For a specific influence, you can also declare the

//methods explicitly and provide additional code there with the standard initialization

//code. You can evaluate the return value.
METHOD FB_Init : BOOL
VAR_INPUT
	bInitRetains : BOOL; // TRUE: the retain variables are initialized (reset warm / reset cold)
	bInCopyCode	 : BOOL; // TRUE: the instance will be copied to the copy code afterward (online change);
END_VAR
_TaskName			 := 'Remove From Group Task';
_TaskId				 := MoverTaskId.REMOVE_FROM_GROUP;
LogSource.SourceName := _TaskName;
LogSource.SourceId	 := _TaskId;
END_METHOD

{attribute 'monitoring':='call'}
PROPERTY IdentInGroup : UDINT
GET
IdentInGroup := _Ident;
END_GET
SET
_Ident := IdentInGroup;
END_SET
END_PROPERTY

METHOD Reset
Executed				  := FALSE;
_Error					  := FALSE;
_ErrorID				  := 0;
_Busy					  := FALSE;
ExecuteWatchdog			  := 0;
_CommandExecuted		  := FALSE;
RemoveFromGroupFb.Execute := FALSE;
END_METHOD

END_FUNCTION_BLOCK

// _Internal/Mover/Tasks/Wrappers/RemoveAxisFromGroup
FUNCTION_BLOCK RemoveAxisFromGroup IMPLEMENTS I_AxisOnGroup
VAR
	_RemoveAxisFromGroup : MC_RemoveAxisFromGroup;
	_Ident				 : UDINT;
END_VAR

VAR_IN_OUT
	AxesGroup : Tc3_McCoordinatedMotion.AXES_GROUP_REF;
END_VAR

_RemoveAxisFromGroup(AxesGroup := AxesGroup);

{attribute 'monitoring':='call'}
PROPERTY Execute : BOOL
GET
Execute := _RemoveAxisFromGroup.Execute;
END_GET
SET
_RemoveAxisFromGroup.Execute := Execute;
END_SET
END_PROPERTY

{attribute 'monitoring':='call'}
PROPERTY IdentInGroup : UDINT
GET
IdentInGroup := _Ident;
END_GET
SET
_Ident := IdentInGroup;
_RemoveAxisFromGroup.IdentInGroup :=UDINT_TO_IDENTINGROUP(IdentInGroup);
END_SET
END_PROPERTY

{attribute 'monitoring':='call'}
PROPERTY Busy : BOOL
GET
Busy := _RemoveAxisFromGroup.Busy;
END_GET
END_PROPERTY

{attribute 'monitoring':='call'}
PROPERTY Done : BOOL
GET
Done := _RemoveAxisFromGroup.Done;
END_GET
END_PROPERTY

{attribute 'monitoring':='call'}
PROPERTY Error : BOOL
GET
Error := _RemoveAxisFromGroup.Error;
END_GET
END_PROPERTY

{attribute 'monitoring':='call'}
PROPERTY ErrorId : UDINT
GET
ErrorId := _RemoveAxisFromGroup.ErrorId;
END_GET
END_PROPERTY

END_FUNCTION_BLOCK

// _Internal/Mover/Tasks/HaltMoverCATask
{attribute 'no_explicit_call' := 'This FB is a CLASS and must be accessed using methods or properties'}
FUNCTION_BLOCK HaltMoverCATask EXTENDS XtsMoverTaskResult IMPLEMENTS I_XtsMoverTask
VAR
	_Axis						: I_AxisRef;
	_BasicDynamics				: I_BaseDynamics;
	_CollisionAvoidanceDynamics : I_CollisionAvoidanceDynamics;
	_DefaultFb					: HaltCa;
	HaltFb						: I_HaltCa := _DefaultFb;
END_VAR

PROPERTY Axis : I_AxisRef
GET
Axis := _Axis;
END_GET
SET
VAR
	Mover : I_XtsMover;
END_VAR
_Axis := Axis;
__QUERYINTERFACE(_Axis, Mover);
__QUERYINTERFACE(Mover.Parameters, _BasicDynamics);
__QUERYINTERFACE(Mover.TracePublisher, _Logger);
__QUERYINTERFACE(Mover.Parameters, _CollisionAvoidanceDynamics);
END_SET
END_PROPERTY

METHOD CyclicLogic
SUPER^.CyclicLogic();			//Watchdog handling
_DefaultFb(Axis := _Axis.Axis); //Call on the default implementation not the interface!!
HaltFb.Execute := FALSE;
_Busy		   := HaltFb.Busy;
IF _Busy THEN
	RETURN;
END_IF

(*Latch signals if they are set by the FB instance itself.
Only reset them in the event of an Task.Execute() call*)
_Error := HaltFb.Error OR _Error;
IF HaltFb.ErrorId <> 0 THEN
	_ErrorID := HaltFb.ErrorId;
END_IF
END_METHOD

METHOD Execute : I_XtsMoverTaskResult
Execute			:= THIS^;
ExecuteWatchdog := ExecuteWatchdog + 1;

//Protect against repeated calls
IF _Busy OR _CommandExecuted THEN
	RETURN;
END_IF

_Error				 := FALSE;
_ErrorID			 := 0;
_Busy				 := TRUE;
HaltFb.Gap			 := _CollisionAvoidanceDynamics.Gap;
HaltFb.Deceleration	 := _BasicDynamics.Deceleration;
HaltFb.Jerk			 := _BasicDynamics.Jerk;
HaltFb.Execute		 := TRUE;
_CommandExecuted	 := TRUE;
LogMessage.Severity	 := 1;
LogMessage.Message	 := CONCAT('Commanded to Halt with Deceleration:', TO_STRING(_BasicDynamics.Deceleration));
LogMessage.MessageId := E_XtsLogMessage.MoverCommandedToHalt;
_Logger.LogMessageInstance(LogSource, LogMessage);
END_METHOD

//FB_Init is always available implicitly and it is used primarily for initialization.

//The return value is not evaluated. For a specific influence, you can also declare the

//methods explicitly and provide additional code there with the standard initialization

//code. You can evaluate the return value.
METHOD FB_Init : BOOL
VAR_INPUT
	bInitRetains : BOOL; // TRUE: the retain variables are initialized (reset warm / reset cold)
	bInCopyCode	 : BOOL; // TRUE: the instance will be copied to the copy code afterward (online change)
END_VAR
_TaskName			 := 'Halt CA';
_TaskId				 := MoverTaskId.HALT_MOVER;
LogSource.SourceName := _TaskName;
LogSource.SourceId	 := _TaskId;
END_METHOD

PROPERTY Interrupted : BOOL
GET
VAR
	Mover : I_XtsMover;
END_VAR
IF NOT  _CommandExecuted THEN
	Interrupted := FALSE;
END_IF

Interrupted := Mover.CurrentTask.TaskName <> 'Halt Mover' AND Mover.CurrentTask.Busy;
END_GET
END_PROPERTY

METHOD Reset
_Error			 := FALSE;
_ErrorID		 := 0;
_Busy			 := FALSE;
ExecuteWatchdog	 := 0;
_CommandExecuted := FALSE;
HaltFb.Execute	 := FALSE;
END_METHOD

END_FUNCTION_BLOCK

// _Internal/Mover/Tasks/Wrappers/HaltCa
FUNCTION_BLOCK HaltCa IMPLEMENTS I_HaltCa
VAR
	_mcHaltCa : MC_HaltCA;
END_VAR

VAR_IN_OUT
	Axis : Tc2_MC2.AXIS_REF;
END_VAR

_mcHaltCa(Axis := Axis);

{attribute 'monitoring':='call'}
PROPERTY Deceleration : MC_LREAL
GET
Deceleration := _mcHaltCa.Deceleration;
END_GET
SET
_mcHaltCa.Deceleration := Deceleration;
END_SET
END_PROPERTY

{attribute 'monitoring':='call'}
PROPERTY Execute : BOOL
GET
Execute := _mcHaltCa.Execute;
END_GET
SET
_mcHaltCa.Execute := Execute;
END_SET
END_PROPERTY

{attribute 'monitoring':='call'}
PROPERTY Gap : MC_LREAL
GET
Gap := _mcHaltCa.Gap;
END_GET
SET
_mcHaltCa.Gap := Gap;
END_SET
END_PROPERTY

{attribute 'monitoring':='call'}
PROPERTY Jerk : MC_LREAL
GET
Jerk := _mcHaltCa.Jerk;
END_GET
SET
_mcHaltCa.Jerk := Jerk;
END_SET
END_PROPERTY

PROPERTY Options : ST_HaltCAOptions
GET
Options := _mcHaltCa.Options;
END_GET
SET
_mcHaltCa.Options := Options;
END_SET
END_PROPERTY

{attribute 'monitoring':='call'}
PROPERTY Active : BOOL
GET
Active := _mcHaltCa.Active;
END_GET
END_PROPERTY

{attribute 'monitoring':='call'}
PROPERTY Busy : BOOL
GET
Busy := _mcHaltCa.Busy;
END_GET
END_PROPERTY

{attribute 'monitoring':='call'}
PROPERTY CommandAborted : BOOL
GET
CommandAborted := _mcHaltCa.CommandAborted;
END_GET
END_PROPERTY

{attribute 'monitoring':='call'}
PROPERTY Done : BOOL
GET
Done := _mcHaltCa.Done;
END_GET
END_PROPERTY

{attribute 'monitoring':='call'}
PROPERTY Error : BOOL
GET
Error := _mcHaltCa.Error;
END_GET
END_PROPERTY

{attribute 'monitoring':='call'}
PROPERTY ErrorId : UDINT
GET
ErrorId := _mcHaltCa.ErrorId;
END_GET
END_PROPERTY

END_FUNCTION_BLOCK

// _Internal/Mover/Tasks/Wrappers/Interfaces/I_HaltCa
INTERFACE I_HaltCa EXTENDS I_BaseCollisionAvoidance

{attribute 'monitoring':='call'}
PROPERTY Deceleration : MC_LREAL
GET
END_GET
SET
END_SET
END_PROPERTY

{attribute 'monitoring':='call'}
PROPERTY Jerk : MC_LREAL
GET
END_GET
SET
END_SET
END_PROPERTY

PROPERTY Options : ST_HaltCAOptions
GET
END_GET
SET
END_SET
END_PROPERTY

{attribute 'monitoring':='call'}
PROPERTY CommandAborted : BOOL
GET
END_GET
END_PROPERTY

END_INTERFACE

// _Internal/Mover/Tasks/Wrappers/Interfaces/I_BaseCollisionAvoidance
INTERFACE I_BaseCollisionAvoidance EXTENDS I_Base

{attribute 'monitoring':='call'}
PROPERTY Execute : BOOL
GET
END_GET
SET
END_SET
END_PROPERTY

{attribute 'monitoring':='call'}
PROPERTY Gap : MC_LREAL
GET
END_GET
SET
END_SET
END_PROPERTY

{attribute 'monitoring':='call'}
PROPERTY Active : BOOL
GET
END_GET
END_PROPERTY

{attribute 'monitoring':='call'}
PROPERTY Busy : BOOL
GET
END_GET
END_PROPERTY

{attribute 'monitoring':='call'}
PROPERTY Error : BOOL
GET
END_GET
END_PROPERTY

{attribute 'monitoring':='call'}
PROPERTY ErrorId : UDINT
GET
END_GET
END_PROPERTY

END_INTERFACE

// _Internal/Mover/Tasks/MoveToPositionCATask
{attribute 'no_explicit_call' := 'This FB is a CLASS and must be accessed using methods or properties'}
FUNCTION_BLOCK MoveToPositionCATask EXTENDS XtsMoverTaskResult IMPLEMENTS I_XtsMoverTask
VAR
	_Axis						: I_AxisRef;
	_DefaultMovePosFb			: ARRAY[0..1] OF MoveToAbsolutePositionCa;
	idx							: DINT := 1; //Start at 1 so that the first call uses 0 (execute changes the index when called)
	MovePosFb					: ARRAY[0..1] OF I_MoveToPositionCA;
	_BasicDyanmics				: I_BaseDynamics;
	_CollisionAvoidanceDynamics : I_CollisionAvoidanceDynamics;
	_DestinationPosition		: I_MoveToPositionParameters;
	_Status						: I_XtsMoverStatus;
END_VAR

PROPERTY Axis : I_AxisRef
GET
Axis := _Axis;
END_GET
SET
VAR
	Mover : I_XtsMover;
END_VAR
_Axis := Axis;
__QUERYINTERFACE(_Axis, Mover);
__QUERYINTERFACE(Mover.Parameters, _BasicDyanmics);
__QUERYINTERFACE(Mover.Parameters, _CollisionAvoidanceDynamics);
__QUERYINTERFACE(Mover.Parameters, _DestinationPosition);
__QUERYINTERFACE(Mover.Status, _Status);
__QUERYINTERFACE(Mover.TracePublisher, _Logger);
END_SET
END_PROPERTY

METHOD CyclicLogic
SUPER^.CyclicLogic(); //Watchdog handling
_DefaultMovePosFb[0](Axis := _Axis.Axis);
_DefaultMovePosFb[1](Axis := _Axis.Axis);
_DefaultMovePosFb[0].Execute := FALSE;
_DefaultMovePosFb[1].Execute := FALSE;
MovePosFb[idx].Execute		 := FALSE;
_Busy						 := MovePosFb[idx].Busy;
IF _Busy THEN
	_Status.CommandedPosition := MovePosFb[idx].Position;
	RETURN;
END_IF

_Error := MovePosFb[idx].Error OR _Error;
IF MovePosFb[idx].ErrorId <> 0 THEN
	_ErrorID := MovePosFb[idx].ErrorId;
END_IF
END_METHOD

METHOD Execute : I_XtsMoverTaskResult
Execute			:= THIS^;
ExecuteWatchdog := ExecuteWatchdog + 1;
IF _CommandExecuted THEN
	RETURN;
END_IF

IF idx = 1 THEN
	idx := 0;
ELSE
	idx := 1;
END_IF

_Error						:= FALSE;
_ErrorId					:= 0;
_Busy						:= TRUE;
MovePosFb[idx].Position		:= _DestinationPosition.Position;
MovePosFb[idx].Velocity		:= _BasicDyanmics.Velocity;
MovePosFb[idx].Acceleration := _BasicDyanmics.Acceleration;
MovePosFb[idx].Deceleration := _BasicDyanmics.Deceleration;
MovePosFb[idx].Jerk			:= _BasicDyanmics.Jerk;
MovePosFb[idx].Direction	:= _BasicDyanmics.Direction;
MovePosFb[idx].Gap			:= _CollisionAvoidanceDynamics.Gap;
MovePosFb[idx].Execute		:= TRUE;
_CommandExecuted			:= TRUE;
LogMessage.Severity			:= 1;
LogMessage.Message			:= CONCAT('Commanded to move to ', TO_STRING(_DestinationPosition.Position));
LogMessage.MessageId		:= E_XtsLogMessage.MoverCommandedToPosition;
_Logger.LogMessageInstance(LogSource, LogMessage);
END_METHOD

//FB_Init is always available implicitly and it is used primarily for initialization.

//The return value is not evaluated. For a specific influence, you can also declare the

//methods explicitly and provide additional code there with the standard initialization

//code. You can evaluate the return value.
METHOD FB_Init : BOOL
VAR_INPUT
	bInitRetains : BOOL; // TRUE: the retain variables are initialized (reset warm / reset cold)
	bInCopyCode	 : BOOL; // TRUE: the instance will be copied to the copy code afterward (online change)
END_VAR
_TaskName			 := 'Move To Position';
MovePosFb[0]		 := _DefaultMovePosFb[0];
MovePosFb[1]		 := _DefaultMovePosFb[1];
_TaskId				 := MoverTaskId.MOVE_TO_POSITION;
LogSource.SourceName := _TaskName;
LogSource.SourceId	 := _TaskId;
END_METHOD

METHOD Reset
_Error				 := FALSE;
_ErrorID			 := 0;
_Busy				 := FALSE;
ExecuteWatchdog		 := 0;
_CommandExecuted	 := FALSE;
MovePosFb[0].Execute := FALSE;
MovePosFb[1].Execute := FALSE;
END_METHOD

END_FUNCTION_BLOCK

// _Internal/Mover/Tasks/Wrappers/MoveToAbsolutePositionCA
FUNCTION_BLOCK MoveToAbsolutePositionCA IMPLEMENTS I_MoveToPositionCA
VAR
	_McMoveAbsoluteFb : MC_MoveAbsoluteCA;
END_VAR

VAR_IN_OUT
	Axis	  : Tc2_Mc2.AXIS_REF;
END_VAR

_McMoveAbsoluteFb(Axis := Axis);

{attribute 'monitoring':='call'}
PROPERTY Acceleration : MC_LREAL
GET
Acceleration := _McMoveAbsoluteFb.Acceleration;
END_GET
SET
_McMoveAbsoluteFb.Acceleration := Acceleration;
END_SET
END_PROPERTY

{attribute 'monitoring':='call'}
PROPERTY BufferMode : Tc3_McCollisionAvoidance.MC_BUFFER_MODE
GET
BufferMode := _McMoveAbsoluteFb.BufferMode;
END_GET
SET
_McMoveAbsoluteFb.BufferMode := BufferMode;
END_SET
END_PROPERTY

{attribute 'monitoring':='call'}
PROPERTY ContinuousUpdate : BOOL
GET
ContinuousUpdate := _McMoveAbsoluteFb.ContinuousUpdate;
END_GET
SET
_McMoveAbsoluteFb.ContinuousUpdate := ContinuousUpdate;
END_SET
END_PROPERTY

{attribute 'monitoring':='call'}
PROPERTY Deceleration : MC_LREAL
GET
Deceleration := _McMoveAbsoluteFb.Deceleration;
END_GET
SET
_McMoveAbsoluteFb.Deceleration := Deceleration;
END_SET
END_PROPERTY

{attribute 'monitoring':='call'}
PROPERTY Direction : Tc3_Mc3Definitions.MC_DIRECTION;
GET
Direction := _McMoveAbsoluteFb.Direction;
END_GET
SET
_McMoveAbsoluteFb.Direction := Direction;
END_SET
END_PROPERTY

{attribute 'monitoring':='call'}
PROPERTY Execute : BOOL
GET
Execute := _McMoveAbsoluteFb.Execute;
END_GET
SET
_McMoveAbsoluteFb.Execute := Execute;
END_SET
END_PROPERTY

{attribute 'monitoring':='call'}
PROPERTY Gap : MC_LREAL
GET
Gap := _McMoveAbsoluteFb.Gap;
END_GET
SET
_McMoveAbsoluteFb.Gap := Gap;
END_SET
END_PROPERTY

{attribute 'monitoring':='call'}
PROPERTY Jerk : MC_LREAL
GET
Jerk := _McMoveAbsoluteFb.Jerk;
END_GET
SET
_McMoveAbsoluteFb.Jerk := Jerk;
END_SET
END_PROPERTY

PROPERTY Options : ST_MoveAbsoluteCAOptions
GET
Options := _McMoveAbsoluteFb.Options;
END_GET
SET
_McMoveAbsoluteFb.Options := Options;
END_SET
END_PROPERTY

{attribute 'monitoring':='call'}
PROPERTY Position : MC_LREAL
GET
Position := _McMoveAbsoluteFb.Position;
END_GET
SET
_McMoveAbsoluteFb.Position := Position;
END_SET
END_PROPERTY

{attribute 'monitoring':='call'}
PROPERTY Velocity : MC_LREAL
GET
Velocity := _McMoveAbsoluteFb.Velocity;
END_GET
SET
_McMoveAbsoluteFb.Velocity := Velocity;
END_SET
END_PROPERTY

{attribute 'monitoring':='call'}
PROPERTY Active : BOOL
GET
Active := _McMoveAbsoluteFb.Active;
END_GET
END_PROPERTY

{attribute 'monitoring':='call'}
PROPERTY Busy : BOOL
GET
Busy := _McMoveAbsoluteFb.Busy;
END_GET
END_PROPERTY

{attribute 'monitoring':='call'}
PROPERTY CommandAborted : BOOL
GET
CommandAborted := _McMoveAbsoluteFb.CommandAborted;
END_GET
END_PROPERTY

{attribute 'monitoring':='call'}
PROPERTY Done : BOOL
GET
Done := _McMoveAbsoluteFb.Done;
END_GET
END_PROPERTY

{attribute 'monitoring':='call'}
PROPERTY Error : BOOL
GET
Error := _McMoveAbsoluteFb.Error;
END_GET
END_PROPERTY

{attribute 'monitoring':='call'}
PROPERTY ErrorId : UDINT
GET
ErrorId := _McMoveAbsoluteFb.ErrorId;
END_GET
END_PROPERTY

END_FUNCTION_BLOCK

// _Internal/Mover/Tasks/Wrappers/Interfaces/I_MoveToPositionCA
INTERFACE I_MoveToPositionCA EXTENDS I_BaseCollisionAvoidance, I_DynamicsCollisionAvoidance

{attribute 'monitoring':='call'}
PROPERTY BufferMode : Tc3_McCollisionAvoidance.MC_BUFFER_MODE
GET
END_GET
SET
END_SET
END_PROPERTY

{attribute 'monitoring':='call'}
PROPERTY ContinuousUpdate : BOOL
GET
END_GET
SET
END_SET
END_PROPERTY

{attribute 'monitoring':='call'}
PROPERTY Direction : Tc3_Mc3Definitions.MC_DIRECTION;
GET
END_GET
SET
END_SET
END_PROPERTY

PROPERTY Options : ST_MoveAbsoluteCAOptions
GET
END_GET
SET
END_SET
END_PROPERTY

{attribute 'monitoring':='call'}
PROPERTY Position : MC_LREAL
GET
END_GET
SET
END_SET
END_PROPERTY

{attribute 'monitoring':='call'}
PROPERTY CommandAborted : BOOL
GET
END_GET
END_PROPERTY

END_INTERFACE

// _Internal/Mover/Tasks/Wrappers/Interfaces/I_DynamicsCollisionAvoidance
INTERFACE I_DynamicsCollisionAvoidance EXTENDS I_BaseCollisionAvoidance

{attribute 'monitoring':='call'}
PROPERTY Acceleration : MC_LREAL
GET
END_GET
SET
END_SET
END_PROPERTY

{attribute 'monitoring':='call'}
PROPERTY Deceleration : MC_LREAL
GET
END_GET
SET
END_SET
END_PROPERTY

{attribute 'monitoring':='call'}
PROPERTY Jerk : MC_LREAL
GET
END_GET
SET
END_SET
END_PROPERTY

{attribute 'monitoring':='call'}
PROPERTY Velocity : MC_LREAL
GET
END_GET
SET
END_SET
END_PROPERTY

{attribute 'monitoring':='call'}
PROPERTY CommandAborted : BOOL
GET
END_GET
END_PROPERTY

END_INTERFACE

// _Internal/Mover/Tasks/MoveVelocityTask
{attribute 'no_explicit_call' := 'This FB is a CLASS and must be accessed using methods or properties'}
FUNCTION_BLOCK MoveVelocityTask EXTENDS XtsMoverTaskResult IMPLEMENTS I_XtsMoverTask
VAR
	_Axis						  : I_AxisRef;
	_XtsMover					  : I_XtsMover;
	_DefaultMovePosFb			  : ARRAY[0..1] OF MoveToRelativePositionCA;
	MoveRelFb					  : ARRAY[0..1] OF I_MoveToPositionCA;
	idx							  : DINT := 1;
	_BasicDynamics				  : I_BaseDynamics;
	_CollisionAvoidanceParameters : I_CollisionAvoidanceDynamics;
END_VAR

PROPERTY Axis : I_AxisRef
GET
Axis := _Axis;
END_GET
SET
_Axis := Axis;
__QUERYINTERFACE(_Axis, _XtsMover);
__QUERYINTERFACE(_XtsMover.Parameters, _BasicDynamics);
__QUERYINTERFACE(_XtsMover.Parameters, _CollisionAvoidanceParameters);
__QUERYINTERFACE(_XtsMover.TracePublisher, _Logger);
END_SET
END_PROPERTY

METHOD CyclicLogic
VAR 
	velocityDifference : LREAL;
END_VAR
SUPER^.CyclicLogic(); //Watchdog handling
_DefaultMovePosFb[0](Axis := _Axis.Axis);
_DefaultMovePosFb[1](Axis := _Axis.Axis);
_DefaultMovePosFb[0].Execute := FALSE;
_DefaultMovePosFb[1].Execute := FALSE;
MoveRelFb[idx].Execute		 := FALSE;
_Busy						 := MoveRelFb[idx].Busy;
IF _Busy AND NOT _XtsMover.InVelocity THEN
	RETURN;
END_IF

_Busy  := FALSE; //Incase we get here from being InVelocity
_Error := MoveRelFb[idx].Error OR _Error;
IF MoveRelFb[idx].ErrorId <> 0 THEN
	_ErrorID := MoveRelFb[idx].ErrorId;
END_IF
END_METHOD

METHOD Execute : I_XtsMoverTaskResult
Execute			:= THIS^;
ExecuteWatchdog := ExecuteWatchdog + 1;
IF _CommandExecuted THEN
	RETURN;
END_IF

IF idx = 1 THEN
	idx := 0;
ELSE
	idx := 1;
END_IF

_Error	 := FALSE;
_ErrorId := 0;
_Busy	 := TRUE;
IF _BasicDynamics.Direction = Tc3_Mc3Definitions.MC_DIRECTION.mcDirectionNegative THEN
	MoveRelFb[idx].Position := -1E10;
ELSE
	MoveRelFb[idx].Position := 1E10;
END_IF

MoveRelFb[idx].Velocity		:= _BasicDynamics.Velocity;
MoveRelFb[idx].Acceleration := _BasicDynamics.Acceleration;
MoveRelFb[idx].Deceleration := _BasicDynamics.Deceleration;
MoveRelFb[idx].Jerk			:= _BasicDynamics.Jerk;
MoveRelFb[idx].Gap			:= _CollisionAvoidanceParameters.Gap;
MoveRelFb[idx].Execute		:= TRUE;
_CommandExecuted			:= TRUE;
LogMessage.Severity			:= 1;
LogMessage.Message			:= CONCAT(CONCAT(CONCAT('Commanded to Move Velocity at ', TO_STRING(_BasicDynamics.Velocity)), ' with Direction '), TO_STRING(_BasicDynamics.Deceleration));
LogMessage.MessageId		:= E_XtsLogMessage.MoverCommandedToMoveVelocity;
_Logger.LogMessageInstance(LogSource, LogMessage);
END_METHOD

//FB_Init is always available implicitly and it is used primarily for initialization.

//The return value is not evaluated. For a specific influence, you can also declare the

//methods explicitly and provide additional code there with the standard initialization

//code. You can evaluate the return value.
METHOD FB_Init : BOOL
VAR_INPUT
	bInitRetains : BOOL; // TRUE: the retain variables are initialized (reset warm / reset cold)
	bInCopyCode	 : BOOL; // TRUE: the instance will be copied to the copy code afterward (online change)
END_VAR
_TaskName			 := 'Move Velocity';
MoveRelFb[0]		 := _DefaultMovePosFb[0];
MoveRelFb[1]		 := _DefaultMovePosFb[1];
_TaskId				 := MoverTaskId.MOVE_VELOCITY;
LogSource.SourceName := _TaskName;
LogSource.SourceId	 := _TaskId;
END_METHOD

METHOD Reset
_Error				 := FALSE;
_ErrorID			 := 0;
_Busy				 := FALSE;
ExecuteWatchdog		 := 0;
_CommandExecuted	 := FALSE;
MoveRelFb[0].Execute := FALSE;
MoveRelFb[1].Execute := FALSE;
END_METHOD

END_FUNCTION_BLOCK

// _Internal/Mover/Tasks/Wrappers/MoveToRelativePositionCA
FUNCTION_BLOCK MoveToRelativePositionCA IMPLEMENTS I_MoveToPositionCA
VAR
	_McMoveRelativeCa : MC_MoveRelativeCA;
END_VAR

VAR_IN_OUT
	Axis	  : Tc2_Mc2.AXIS_REF;
END_VAR

_McMoveRelativeCa(Axis := Axis);

{attribute 'monitoring':='call'}
PROPERTY Acceleration : MC_LREAL
GET
Acceleration := _McMoveRelativeCa.Acceleration;
END_GET
SET
_McMoveRelativeCa.Acceleration := Acceleration;
END_SET
END_PROPERTY

{attribute 'monitoring':='call'}
PROPERTY BufferMode : Tc3_McCollisionAvoidance.MC_BUFFER_MODE
GET
BufferMode := _McMoveRelativeCa.BufferMode;
END_GET
SET
_McMoveRelativeCa.BufferMode := BufferMode;
END_SET
END_PROPERTY

{attribute 'monitoring':='call'}
PROPERTY ContinuousUpdate : BOOL
GET
ContinuousUpdate := _McMoveRelativeCa.ContinuousUpdate;
END_GET
SET
_McMoveRelativeCa.ContinuousUpdate := ContinuousUpdate;
END_SET
END_PROPERTY

{attribute 'monitoring':='call'}
PROPERTY Deceleration : MC_LREAL
GET
Deceleration := _McMoveRelativeCa.Deceleration;
END_GET
SET
_McMoveRelativeCa.Deceleration := Deceleration;
END_SET
END_PROPERTY

{attribute 'monitoring':='call'}
PROPERTY Direction : Tc3_Mc3Definitions.MC_DIRECTION;
GET
END_GET
SET
//TODO - create interface for relative that doesn't include direction for simplification
END_SET
END_PROPERTY

{attribute 'monitoring':='call'}
PROPERTY Execute : BOOL
GET
Execute := _McMoveRelativeCa.Execute;
END_GET
SET
_McMoveRelativeCa.Execute := Execute;
END_SET
END_PROPERTY

{attribute 'monitoring':='call'}
PROPERTY Gap : MC_LREAL
GET
Gap := _McMoveRelativeCa.Gap;
END_GET
SET
_McMoveRelativeCa.Gap := Gap;
END_SET
END_PROPERTY

{attribute 'monitoring':='call'}
PROPERTY Jerk : MC_LREAL
GET
Jerk := _McMoveRelativeCa.Jerk;
END_GET
SET
_McMoveRelativeCa.Jerk := Jerk;
END_SET
END_PROPERTY

PROPERTY Options : ST_MoveAbsoluteCAOptions
GET
//Options := _McMoveRelativeCa.Options;
END_GET
SET
//_McMoveRelativeCa.Options := Options;
END_SET
END_PROPERTY

{attribute 'monitoring':='call'}
PROPERTY Position : MC_LREAL
GET
Position := _McMoveRelativeCa.Distance;
END_GET
SET
_McMoveRelativeCa.Distance := Position;
END_SET
END_PROPERTY

{attribute 'monitoring':='call'}
PROPERTY Velocity : MC_LREAL
GET
Velocity := _McMoveRelativeCa.Velocity;
END_GET
SET
_McMoveRelativeCa.Velocity := Velocity;
END_SET
END_PROPERTY

{attribute 'monitoring':='call'}
PROPERTY Active : BOOL
GET
Active := _McMoveRelativeCa.Active;
END_GET
END_PROPERTY

{attribute 'monitoring':='call'}
PROPERTY Busy : BOOL
GET
Busy := _McMoveRelativeCa.Busy;
END_GET
END_PROPERTY

{attribute 'monitoring':='call'}
PROPERTY CommandAborted : BOOL
GET
CommandAborted := _McMoveRelativeCa.CommandAborted;
END_GET
END_PROPERTY

{attribute 'monitoring':='call'}
PROPERTY Done : BOOL
GET
Done := _McMoveRelativeCa.Done;
END_GET
END_PROPERTY

{attribute 'monitoring':='call'}
PROPERTY Error : BOOL
GET
Error := _McMoveRelativeCa.Error;
END_GET
END_PROPERTY

{attribute 'monitoring':='call'}
PROPERTY ErrorId : UDINT
GET
ErrorId := _McMoveRelativeCa.ErrorId;
END_GET
END_PROPERTY

END_FUNCTION_BLOCK

// _Internal/Mover/Tasks/MoveToStationTask
{attribute 'no_explicit_call' := 'This FB is a CLASS and must be accessed using methods or properties'}
FUNCTION_BLOCK MoveToStationTask EXTENDS XtsMoverTaskResult IMPLEMENTS I_MoveToStationTask, I_Cyclic
VAR
	_Axis						: I_AxisRef;
	_DefaultMovePosFb			: ARRAY[0..1] OF MoveToAbsolutePositionCa;
	MovePosFb					: ARRAY[0..1] OF I_MoveToPositionCA;
	idx							: DINT := 1;
	_BasicDyanmics				: I_BaseDynamics;
	_CollisionAvoidanceDynamics : I_CollisionAvoidanceDynamics;
	_DestinationPosition		: I_MoveToPositionParameters;
	_Station					: I_XtsStation;
	_Status						: I_XtsMoverStatus;
END_VAR

PROPERTY Axis : I_AxisRef
GET
Axis := _Axis;
END_GET
SET
VAR
	Mover : I_XtsMover;
END_VAR
_Axis := Axis;
__QUERYINTERFACE(_Axis, Mover);
__QUERYINTERFACE(Mover.Parameters, _BasicDyanmics);
__QUERYINTERFACE(Mover.Parameters, _CollisionAvoidanceDynamics);
__QUERYINTERFACE(Mover.Parameters, _DestinationPosition);
__QUERYINTERFACE(Mover.Status, _Status);
__QUERYINTERFACE(Mover.TracePublisher, _Logger);
END_SET
END_PROPERTY

METHOD CyclicLogic
SUPER^.CyclicLogic(); //Watchdog handling
_DefaultMovePosFb[0](Axis := _Axis.Axis);
_DefaultMovePosFb[1](Axis := _Axis.Axis);
_DefaultMovePosFb[0].Execute := FALSE;
_DefaultMovePosFb[1].Execute := FALSE;
MovePosFb[idx].Execute		 := FALSE;
_Busy						 := MovePosFb[idx].Busy;
IF _Busy THEN
	RETURN;
END_IF

_Error := MovePosFb[idx].Error OR _Error;
IF MovePosFb[idx].ErrorId <> 0 THEN
	_ErrorID := MovePosFb[idx].ErrorId;
END_IF
END_METHOD

METHOD Execute : I_XtsMoverTaskResult
VAR
	Mover		 : I_XtsMover;
	_StationName : T_MaxString;
END_VAR
Execute			:= THIS^;
ExecuteWatchdog := ExecuteWatchdog + 1;
IF _CommandExecuted THEN
	RETURN;
END_IF

IF idx = 1 THEN
	idx := 0;
ELSE
	idx := 1;
END_IF

_Error						  := FALSE;
_ErrorId					  := 0;
_Busy						  := TRUE;
_DestinationPosition.Position := _Station.Position;
MovePosFb[idx].Position		  := _DestinationPosition.Position;
MovePosFb[idx].Velocity		  := _BasicDyanmics.Velocity;
MovePosFb[idx].Acceleration	  := _BasicDyanmics.Acceleration;
MovePosFb[idx].Deceleration	  := _BasicDyanmics.Deceleration;
MovePosFb[idx].Jerk			  := _BasicDyanmics.Jerk;
MovePosFb[idx].Direction	  := _BasicDyanmics.Direction;
MovePosFb[idx].Gap			  := _CollisionAvoidanceDynamics.Gap;
__QUERYINTERFACE(_Axis, Mover);
_Station.RegisterMover(Mover);
_Status.CommandedPosition := _Station.Position;
_Status.CommandedStation  := _Station;
MovePosFb[idx].Execute	   := TRUE;
_CommandExecuted		   := TRUE;
_StationName			   := _Station.Name;
LogMessage.Severity		   := 1;
LogMessage.Message		   := CONCAT('Commanded to move to ', _StationName);
LogMessage.MessageId	   := E_XtsLogMessage.MoverCommandedToStation;
_Logger.LogMessageInstance(LogSource, LogMessage);
END_METHOD

//FB_Init is always available implicitly and it is used primarily for initialization.

//The return value is not evaluated. For a specific influence, you can also declare the

//methods explicitly and provide additional code there with the standard initialization

//code. You can evaluate the return value.
METHOD FB_Init : BOOL
VAR_INPUT
	bInitRetains : BOOL; // TRUE: the retain variables are initialized (reset warm / reset cold)
	bInCopyCode	 : BOOL; // TRUE: the instance will be copied to the copy code afterward (online change)
END_VAR
_TaskName			 := 'Move To Station Task';
MovePosFb[0]		 := _DefaultMovePosFb[0];
MovePosFb[1]		 := _DefaultMovePosFb[1];
_TaskId				 := MoverTaskId.MOVE_TO_STATION;
LogSource.SourceName := _TaskName;
LogSource.SourceId	 := _TaskId;
END_METHOD

METHOD Reset
_Error				 := FALSE;
_ErrorID			 := 0;
_Busy				 := FALSE;
ExecuteWatchdog		 := 0;
_CommandExecuted	 := FALSE;
MovePosFb[0].Execute := FALSE;
MovePosFb[1].Execute := FALSE;
END_METHOD

{attribute 'monitoring' := 'call'}
PROPERTY Station : I_XtsStation
GET
Station := _Station;
END_GET
SET
_Station := Station;
END_SET
END_PROPERTY

END_FUNCTION_BLOCK

// _Internal/Mover/Tasks/Interfaces/I_MoveToStationTask
INTERFACE I_MoveToStationTask EXTENDS I_XtsMoverTask, I_MoveToStationParameters

END_INTERFACE

// _Internal/Mover/Tasks/ActivateTrackTask
{attribute 'no_explicit_call' := 'This FB is a CLASS and must be accessed using methods or properties'}
FUNCTION_BLOCK ActivateTrackTask EXTENDS XtsMoverTaskResult IMPLEMENTS I_TakesTrackId, I_XtsMoverTask
VAR
	_Axis				  : I_AxisRef;
	_DefaultActivateTrack : ActivateTrack;
	_ActivateTrack		  : I_ActivateTrack := _DefaultActivateTrack;
	_DesiredTrackId		  : UDINT;
	_DesiredTrack		  : I_XtsTrack := NullObjects.XtsTrack;
	_TrackCollection	  : I_XtsTrackCollection;
	_Status				  : I_XtsMoverStatus;
	Executed			  : BOOL;
END_VAR

PROPERTY Axis : I_AxisRef
GET
Axis := _Axis;
END_GET
SET
_Axis := Axis;
__QUERYINTERFACE(_Axis, _Mover);
__QUERYINTERFACE(_Mover.TracePublisher, _Logger);
__QUERYINTERFACE(_Mover.Status, _Status);
_TrackCollection := _Mover.Tracks;
END_SET
END_PROPERTY

METHOD CyclicLogic
VAR
END_VAR
SUPER^.CyclicLogic(); //Watchdog handling
_DefaultActivateTrack(Axis := _Axis.Axis);
_ActivateTrack.Execute := FALSE;
_Busy				   := _ActivateTrack.Busy;
IF _Busy THEN
	RETURN;
END_IF

(*Latch signals if they are set by the FB instance itself.
Only reset them in the event of an Task.Execute() call*)
IF Executed AND _DesiredTrack <> _Status.CurrentTrack THEN
	Executed			  := FALSE;
	_Status.CurrentTrack := _DesiredTrack;
END_IF

_Error := _ActivateTrack.Error OR _Error;
IF _ActivateTrack.ErrorId <> 0 THEN
	_ErrorID := _ActivateTrack.ErrorId;
END_IF
END_METHOD

METHOD Execute : I_XtsMoverTaskResult
Execute			:= THIS^;
ExecuteWatchdog := ExecuteWatchdog + 1;
//Protect against repeated calls
IF _Busy OR _CommandExecuted THEN
	RETURN;
END_IF

_DesiredTrack		   := _TrackCollection.GetById(_DesiredTrackId);
_ActivateTrack.TrackId := _DesiredTrack.Otcid;
LogMessage.Severity	   := 1;
LogMessage.Message	   := CONCAT('Commanded to Activate Track ', TO_STRING(_DesiredTrack.Otcid));
LogMessage.MessageId   := E_XtsLogMessage.MoverCommandedToActivateTrack;
_Logger.LogMessageInstance(LogSource, LogMessage);
IF _Mover.VirtualMover OR NOT _Mover.Status.MoverInGroup THEN
	_Busy				  := FALSE;
	_Error				  := FALSE;
	_ErrorId			  := 0;
	_Status.CurrentTrack := _DesiredTrack;
	RETURN;
END_IF

_Error				   := FALSE;
_ErrorID			   := 0;
_Busy				   := TRUE;
_ActivateTrack.Execute := TRUE;
Executed			   := TRUE;
_CommandExecuted	   := TRUE;
END_METHOD

//FB_Init is always available implicitly and it is used primarily for initialization.

//The return value is not evaluated. For a specific influence, you can also declare the

//methods explicitly and provide additional code there with the standard initialization

//code. You can evaluate the return value.
METHOD FB_Init : BOOL
VAR_INPUT
	bInitRetains : BOOL; // TRUE: the retain variables are initialized (reset warm / reset cold)
	bInCopyCode	 : BOOL; // TRUE: the instance will be copied to the copy code afterward (online change)
END_VAR
_TaskName			 := 'Activate Track';
_TaskId				 := MoverTaskId.ACTIVATE_TRACK;
LogSource.SourceName := 'Activate Track';
LogSource.SourceId	 := _TaskId;
END_METHOD

METHOD Reset
Executed			   := FALSE;
_Error				   := FALSE;
_ErrorID			   := 0;
_Busy				   := FALSE;
ExecuteWatchdog		   := 0;
_CommandExecuted	   := FALSE;
_ActivateTrack.Execute := FALSE;
END_METHOD

PROPERTY TrackId : UDINT
SET
_DesiredTrackId := TrackId;
END_SET
END_PROPERTY

END_FUNCTION_BLOCK

// _Internal/Mover/Tasks/Interfaces/I_TakesTrackId
INTERFACE I_TakesTrackId EXTENDS I_Base

PROPERTY TrackId : UDINT
SET
END_SET
END_PROPERTY

END_INTERFACE

// _Internal/Mover/Tasks/ResetAxisTask
{attribute 'no_explicit_call' := 'This FB is a CLASS and must be accessed using methods or properties'}
FUNCTION_BLOCK ResetAxisTask EXTENDS XtsMoverTaskResult IMPLEMENTS I_XtsMoverTask
VAR
	_Axis			: I_AxisRef;
	_DefaultResetFb : ResetMover;
	ResetMoverFb	: I_ResetAxis := _DefaultResetFb;
END_VAR

PROPERTY Axis : I_AxisRef
GET
Axis := _Axis;
END_GET
SET
_Axis := Axis;
__QUERYINTERFACE(_Axis, _Mover);
__QUERYINTERFACE(_Mover.TracePublisher, _Logger);
END_SET
END_PROPERTY

METHOD CyclicLogic
VAR
END_VAR
SUPER^.CyclicLogic(); //Watchdog handling
_DefaultResetFb(Axis := _Axis.Axis);
ResetMoverFb.Execute := FALSE;
_Busy				 := ResetMoverFb.Busy;
IF _Busy THEN
	RETURN;
END_IF

(*Latch signals if they are set by the FB instance itself.
Only reset them in the event of an Task.Execute() call*)
_Error := ResetMoverFb.Error OR _Error;
IF ResetMoverFb.ErrorId <> 0 THEN
	_ErrorID := ResetMoverFb.ErrorId;
END_IF
END_METHOD

METHOD Execute : I_XtsMoverTaskResult
Execute			:= THIS^;
ExecuteWatchdog := ExecuteWatchdog + 1;

//Protect against repeated calls
IF _Busy OR _CommandExecuted THEN
	RETURN;
END_IF

LogMessage.Severity	   := 1;
LogMessage.Message	   := 'Commanded to Reset';
LogMessage.MessageId   := E_XtsLogMessage.MoverCommandedToReset;
_Logger.LogMessageInstance(LogSource, LogMessage);

_Error				 := FALSE;
_ErrorID			 := 0;
_Busy				 := TRUE;
ResetMoverFb.Execute := TRUE;
_CommandExecuted	 := TRUE;
END_METHOD

//FB_Init is always available implicitly and it is used primarily for initialization.

//The return value is not evaluated. For a specific influence, you can also declare the

//methods explicitly and provide additional code there with the standard initialization

//code. You can evaluate the return value.
METHOD FB_Init : BOOL
VAR_INPUT
	bInitRetains : BOOL; // TRUE: the retain variables are initialized (reset warm / reset cold)
	bInCopyCode	 : BOOL; // TRUE: the instance will be copied to the copy code afterward (online change)
END_VAR
_TaskName := 'Reset Mover';
_TaskId	  := MoverTaskId.RESET_MOVER;
END_METHOD

METHOD Reset
_Error				 := FALSE;
_ErrorID			 := 0;
_Busy				 := FALSE;
ExecuteWatchdog		 := 0;
_CommandExecuted	 := FALSE;
ResetMoverFb.Execute := FALSE;
END_METHOD

END_FUNCTION_BLOCK

// _Internal/Mover/Tasks/Wrappers/ResetMover
FUNCTION_BLOCK ResetMover IMPLEMENTS I_ResetAxis
VAR
	_McReset : MC_Reset;
END_VAR

VAR_IN_OUT
	Axis : Tc2_Mc2.AXIS_REF;
END_VAR

_McReset(Axis := Axis);

{attribute 'monitoring':='call'}
PROPERTY Execute : BOOL
GET
Execute := _McReset.Execute;
END_GET
SET
_McReset.Execute := Execute;
END_SET
END_PROPERTY

{attribute 'monitoring':='call'}
PROPERTY Busy : BOOL
GET
Busy := _McReset.Busy;
END_GET
END_PROPERTY

{attribute 'monitoring':='call'}
PROPERTY Done : BOOL
GET
Done := _McReset.Done;
END_GET
END_PROPERTY

{attribute 'monitoring':='call'}
PROPERTY Error : BOOL
GET
Error := _McReset.Error;
END_GET
END_PROPERTY

{attribute 'monitoring':='call'}
PROPERTY ErrorId : UDINT
GET
ErrorId := _McReset.ErrorId;
END_GET
END_PROPERTY

END_FUNCTION_BLOCK

// _Internal/Mover/Tasks/Wrappers/Interfaces/I_ResetAxis
INTERFACE I_ResetAxis EXTENDS I_Base

{attribute 'monitoring':='call'}
PROPERTY Execute : BOOL
GET
END_GET
SET
END_SET
END_PROPERTY

{attribute 'monitoring':='call'}
PROPERTY Busy : BOOL
GET
END_GET
END_PROPERTY

{attribute 'monitoring':='call'}
PROPERTY Error : BOOL
GET
END_GET
END_PROPERTY

{attribute 'monitoring':='call'}
PROPERTY ErrorId : UDINT
GET
END_GET
END_PROPERTY

END_INTERFACE

// _Internal/Mover/Tasks/SyncToAxisTask
{attribute 'no_explicit_call' := 'This FB is a CLASS and must be accessed using methods or properties'}
FUNCTION_BLOCK SyncToAxisTask EXTENDS XtsMoverTaskResult IMPLEMENTS I_XtsMoverTask
VAR
	_Axis						  : I_AxisRef;
	_MasterAxis					  : REFERENCE TO AXIS_REF;
	_DefaultFb					  : ARRAY[0..1] OF GearInPosCa;
	GearPosFb					  : ARRAY[0..1] OF I_GearInPosCA;
	idx							  : DINT := 1;
	_BasicDynamics				  : I_BaseDynamics;
	_CollisionAvoidanceParameters : I_CollisionAvoidanceDynamics;
	_SyncAxisParameters			  : I_ContainSyncAxisParameters;
	_Status						  : I_XtsMoverStatus;
END_VAR

PROPERTY Axis : I_AxisRef
GET
Axis := _Axis;
END_GET
SET
VAR
	Mover : I_XtsMover;
END_VAR
_Axis := Axis;
__QUERYINTERFACE(_Axis, Mover);
__QUERYINTERFACE(Mover.Parameters, _BasicDynamics);
__QUERYINTERFACE(Mover.Parameters, _CollisionAvoidanceParameters);
__QUERYINTERFACE(Mover.Parameters, _SyncAxisParameters);
__QUERYINTERFACE(Mover.Status, _Status);
__QUERYINTERFACE(Mover.TracePublisher, _Logger);
END_SET
END_PROPERTY

METHOD CyclicLogic
VAR 
	velocityDifference : LREAL;
END_VAR
SUPER^.CyclicLogic(); //Watchdog handling
_DefaultFb[0](SlaveAxis := _Axis.Axis, MasterAxis := _MasterAxis);
_DefaultFb[1](SlaveAxis := _Axis.Axis, MasterAxis := _MasterAxis);
_DefaultFb[0].Execute  := FALSE;
_DefaultFb[1].Execute  := FALSE;
GearPosFb[idx].Execute := FALSE;
_Busy				   := GearPosFb[idx].Busy;
_Status.InSync		   := GearPosFb[idx].InSync;
IF _Busy AND NOT GearPosFb[idx].InSync THEN
	RETURN;
END_IF

_Error := GearPosFb[idx].Error OR _Error;
IF GearPosFb[idx].ErrorId <> 0 THEN
	_ErrorID := GearPosFb[idx].ErrorId;
END_IF
END_METHOD

METHOD Execute : I_XtsMoverTaskResult
Execute			:= THIS^;
ExecuteWatchdog := ExecuteWatchdog + 1;
IF _CommandExecuted THEN
	RETURN;
END_IF

IF idx = 1 THEN
	idx := 0;
ELSE
	idx := 1;
END_IF

_Error							   := FALSE;
_ErrorId						   := 0;
_Busy							   := TRUE;
_MasterAxis						   REF= _SyncAxisParameters.SyncAxis.MasterAxis;
GearPosFb[idx].Velocity			   := _BasicDynamics.Velocity;
GearPosFb[idx].Acceleration		   := _BasicDynamics.Acceleration;
GearPosFb[idx].Deceleration		   := _BasicDynamics.Deceleration;
GearPosFb[idx].Jerk				   := _BasicDynamics.Jerk;
GearPosFb[idx].Gap				   := _CollisionAvoidanceParameters.Gap;
GearPosFb[idx].MasterSyncPosition  := _SyncAxisParameters.SyncAxis.MasterSyncPosition;
GearPosFb[idx].SlaveSyncPosition   := _SyncAxisParameters.SyncAxis.SlaveSyncPosition;
GearPosFb[idx].MasterStartDistance := _SyncAxisParameters.SyncAxis.MasterStartDistance;
GearPosFb[idx].RatioNumerator	   := _SyncAxisParameters.SyncAxis.RatioNumerator;
GearPosFb[idx].RatioDenominator	   := _SyncAxisParameters.SyncAxis.RatioDenominator;
GearPosFb[idx].SyncStrategy		   := _SyncAxisParameters.SyncAxis.SyncStrategy;
GearPosFb[idx].SyncMode			   := _SyncAxisParameters.SyncAxis.SyncMode;
GearPosFb[idx].Options			   := _SyncAxisParameters.SyncAxis.Options_CA;
GearPosFb[idx].Execute			   := TRUE;
_CommandExecuted				   := TRUE;
LogMessage.Severity				   := 1;
LogMessage.Message				   := 'Commanded to Sync to Axis';
LogMessage.MessageId			   := E_XtsLogMessage.MoverCommandedToSyncAxis;
_Logger.LogMessageInstance(LogSource, LogMessage);
END_METHOD

//FB_Init is always available implicitly and it is used primarily for initialization.

//The return value is not evaluated. For a specific influence, you can also declare the

//methods explicitly and provide additional code there with the standard initialization

//code. You can evaluate the return value.
METHOD FB_Init : BOOL
VAR_INPUT
	bInitRetains : BOOL; // TRUE: the retain variables are initialized (reset warm / reset cold)
	bInCopyCode	 : BOOL; // TRUE: the instance will be copied to the copy code afterward (online change)
END_VAR
_TaskName			 := 'Sync To Axis';
GearPosFb[0]		 := _DefaultFb[0];
GearPosFb[1]		 := _DefaultFb[1];
_TaskId				 := MoverTaskId.SYNC_TO_AXIS;
LogSource.SourceName := _TaskName;
LogSource.SourceId	 := _TaskId;
END_METHOD

METHOD Reset
_Error				 := FALSE;
_ErrorID			 := 0;
_Busy				 := FALSE;
ExecuteWatchdog		 := 0;
_CommandExecuted	 := FALSE;
GearPosFb[0].Execute := FALSE;
GearPosFb[0].Execute := FALSE;
idx					 := 1;
END_METHOD

END_FUNCTION_BLOCK

// _Internal/Mover/Tasks/Wrappers/GearInPosCa
FUNCTION_BLOCK GearInPosCa IMPLEMENTS I_GearInPosCA
VAR
	_Mc_GearInPosCa : MC_GearInPosCA;
END_VAR

VAR_IN_OUT
	MasterAxis : Tc2_Mc2.AXIS_REF;
	SlaveAxis  : Tc2_Mc2.AXIS_REF;
END_VAR

_Mc_GearInPosCa(Master := MasterAxis, Slave := SlaveAxis);

{attribute 'monitoring' := 'call'}
PROPERTY Acceleration : MC_LREAL
GET
Acceleration := _Mc_GearInPosCa.Acceleration;
END_GET
SET
_Mc_GearInPosCa.Acceleration := Acceleration;
END_SET
END_PROPERTY

{attribute 'monitoring' := 'call'}
PROPERTY BufferMode : Tc3_McCollisionAvoidance.MC_BUFFER_MODE
GET
BufferMode := _Mc_GearInPosCa.BufferMode;
END_GET
SET
_Mc_GearInPosCa.BufferMode := BufferMode;
END_SET
END_PROPERTY

{attribute 'monitoring' := 'call'}
PROPERTY ContinuousUpdate : BOOL
GET
ContinuousUpdate := _Mc_GearInPosCa.ContinuousUpdate;
END_GET
SET
_Mc_GearInPosCa.ContinuousUpdate := ContinuousUpdate;
END_SET
END_PROPERTY

{attribute 'monitoring' := 'call'}
PROPERTY Deceleration : MC_LREAL
GET
Deceleration := _Mc_GearInPosCa.Deceleration;
END_GET
SET
_Mc_GearInPosCa.Deceleration := Deceleration;
END_SET
END_PROPERTY

{attribute 'monitoring' := 'call'}
PROPERTY Execute : BOOL
GET
Execute := _Mc_GearInPosCa.Execute;
END_GET
SET
_Mc_GearInPosCa.Execute := Execute;
END_SET
END_PROPERTY

{attribute 'monitoring' := 'call'}
PROPERTY Gap : MC_LREAL
GET
Gap := _Mc_GearInPosCa.Gap;
END_GET
SET
_Mc_GearInPosCa.Gap := Gap;
END_SET
END_PROPERTY

{attribute 'monitoring' := 'call'}
PROPERTY Jerk : MC_LREAL
GET
Jerk := _Mc_GearInPosCa.Jerk;
END_GET
SET
_Mc_GearInPosCa.Jerk := Jerk;
END_SET
END_PROPERTY

{attribute 'monitoring' := 'call'}
PROPERTY MasterStartDistance : MC_LREAL
GET
MasterStartDistance := _Mc_GearInPosCa.MasterStartDistance;
END_GET
SET
_Mc_GearInPosCa.MasterStartDistance := MasterStartDistance;
END_SET
END_PROPERTY

{attribute 'monitoring' := 'call'}
PROPERTY MasterSyncPosition : MC_LREAL
GET
MasterSyncPosition := _Mc_GearInPosCa.MasterSyncPosition;
END_GET
SET
_Mc_GearInPosCa.MasterSyncPosition := MasterSyncPosition;
END_SET
END_PROPERTY

PROPERTY Options : Tc3_McCollisionAvoidance.ST_GearInPosCAOptions
GET
Options := _Mc_GearInPosCa.Options;
END_GET
SET
_Mc_GearInPosCa.Options := Options;
END_SET
END_PROPERTY

{attribute 'monitoring' := 'call'}
PROPERTY RatioDenominator : UINT
GET
RatioDenominator := _Mc_GearInPosCa.RatioDenumerator;
END_GET
SET
_Mc_GearInPosCa.RatioDenumerator := RatioDenominator;
END_SET
END_PROPERTY

{attribute 'monitoring' := 'call'}
PROPERTY RatioNumerator : MC_LREAL
GET
RatioNumerator := _Mc_GearInPosCa.RatioNumerator;
END_GET
SET
_Mc_GearInPosCa.RatioNumerator := RatioNumerator;
END_SET
END_PROPERTY

{attribute 'monitoring' := 'call'}
PROPERTY SlaveSyncPosition : LREAL
GET
SlaveSyncPosition := _Mc_GearInPosCa.SlaveSyncPosition;
END_GET
SET
_Mc_GearInPosCa.SlaveSyncPosition := SlaveSyncPosition;
END_SET
END_PROPERTY

{attribute 'monitoring' := 'call'}
PROPERTY SyncMode : Tc3_McCollisionAvoidance.MC_SYNC_MODE
GET
SyncMode := _Mc_GearInPosCa.SyncMode;
END_GET
SET
_Mc_GearInPosCa.SyncMode := SyncMode;
END_SET
END_PROPERTY

{attribute 'monitoring' := 'call'}
PROPERTY SyncStrategy : Tc3_McCollisionAvoidance.MC_SYNC_STRATEGY
GET
SyncStrategy := _Mc_GearInPosCa.SyncStrategy;
END_GET
SET
_Mc_GearInPosCa.SyncStrategy := SyncStrategy;
END_SET
END_PROPERTY

{attribute 'monitoring' := 'call'}
PROPERTY Velocity : MC_LREAL
GET
Velocity := _Mc_GearInPosCa.Velocity;
END_GET
SET
_Mc_GearInPosCa.Velocity := Velocity;
END_SET
END_PROPERTY

{attribute 'monitoring' := 'call'}
PROPERTY Active : BOOL
GET
Active := _Mc_GearInPosCa.Active;
END_GET
END_PROPERTY

{attribute 'monitoring' := 'call'}
PROPERTY Busy : BOOL
GET
Busy := _Mc_GearInPosCa.Busy;
END_GET
END_PROPERTY

{attribute 'monitoring' := 'call'}
PROPERTY CommandAborted : BOOL
GET
CommandAborted := _Mc_GearInPosCa.CommandAborted;
END_GET
END_PROPERTY

{attribute 'monitoring' := 'call'}
PROPERTY Done : BOOL
GET
END_GET
END_PROPERTY

{attribute 'monitoring' := 'call'}
PROPERTY Error : BOOL
GET
Error := _Mc_GearInPosCa.Error;
END_GET
END_PROPERTY

{attribute 'monitoring' := 'call'}
PROPERTY ErrorId : UDINT
GET
ErrorId := _Mc_GearInPosCa.ErrorId;
END_GET
END_PROPERTY

{attribute 'monitoring' := 'call'}
PROPERTY InSync : BOOL
GET
InSync := _Mc_GearInPosCa.InSync;
END_GET
END_PROPERTY

{attribute 'monitoring' := 'call'}
PROPERTY StartSync : BOOL
GET
StartSync := _Mc_GearInPosCa.StartSync;
END_GET
END_PROPERTY

END_FUNCTION_BLOCK

// _Internal/Mover/Tasks/Wrappers/Interfaces/I_GearInPosCA
INTERFACE I_GearInPosCA EXTENDS I_BaseCollisionAvoidance, I_DynamicsCollisionAvoidance

{attribute 'monitoring' := 'call'}
PROPERTY BufferMode : Tc3_McCollisionAvoidance.MC_BUFFER_MODE
GET
END_GET
SET
END_SET
END_PROPERTY

{attribute 'monitoring' := 'call'}
PROPERTY ContinuousUpdate : BOOL
GET
END_GET
SET
END_SET
END_PROPERTY

{attribute 'monitoring' := 'call'}
PROPERTY MasterStartDistance : MC_LREAL
GET
END_GET
SET
END_SET
END_PROPERTY

{attribute 'monitoring' := 'call'}
PROPERTY MasterSyncPosition : MC_LREAL
GET
END_GET
SET
END_SET
END_PROPERTY

PROPERTY Options : Tc3_McCollisionAvoidance.ST_GearInPosCAOptions
GET
END_GET
SET
END_SET
END_PROPERTY

{attribute 'monitoring' := 'call'}
PROPERTY RatioDenominator : UINT
GET
END_GET
SET
END_SET
END_PROPERTY

{attribute 'monitoring' := 'call'}
PROPERTY RatioNumerator : MC_LREAL
GET
END_GET
SET
END_SET
END_PROPERTY

{attribute 'monitoring' := 'call'}
PROPERTY SlaveSyncPosition : LREAL
GET
END_GET
SET
END_SET
END_PROPERTY

{attribute 'monitoring' := 'call'}
PROPERTY SyncMode : Tc3_McCollisionAvoidance.MC_SYNC_MODE
GET
END_GET
SET
END_SET
END_PROPERTY

{attribute 'monitoring' := 'call'}
PROPERTY SyncStrategy : Tc3_McCollisionAvoidance.MC_SYNC_STRATEGY
GET
END_GET
SET
END_SET
END_PROPERTY

{attribute 'monitoring' := 'call'}
PROPERTY InSync : BOOL
GET
END_GET
END_PROPERTY

{attribute 'monitoring' := 'call'}
PROPERTY StartSync : BOOL
GET
END_GET
END_PROPERTY

END_INTERFACE

// Logging/XtsLocalLogger
{attribute 'hide_all_locals'}
FUNCTION_BLOCK XtsLocalLogger IMPLEMENTS I_XtsLocalLogger
VAR
	_LogEntries : ARRAY[0..XtsCoreParameters.MAX_NUMBER_LOCAL_LOG - 1] OF XtsLogCommand;
	_Entries	: ARRAY[0..XtsCoreParameters.MAX_NUMBER_LOCAL_LOG - 1] OF I_XtsLogCommand;
	_SimpleLog	: ARRAY[0..XtsCoreParameters.MAX_NUMBER_LOCAL_LOG - 1] OF T_MaxString;
END_VAR

METHOD Clear
VAR
	i : UDINT;
END_VAR
FOR i := 0 TO XtsCoreParameters.MAX_NUMBER_LOCAL_LOG - 1 DO
	_LogEntries[i].Arguments  := 0;
	_LogEntries[i].Message	  := '';
	_LogEntries[i].MessageId  := 0;
	_LogEntries[i].TimeStamp  := 0;
	_LogEntries[i].SourceId	  := 0;
	_LogEntries[i].SourceName := '';
END_FOR
END_METHOD

{attribute 'monitoring':='call'}
PROPERTY Commands : REFERENCE TO ARRAY[0..XtsCoreParameters.MAX_NUMBER_LOCAL_LOG - 1] OF T_MaxString
GET
Commands REF= _SimpleLog;
END_GET
END_PROPERTY

{attribute 'monitoring':='call'}
PROPERTY DetailedCommands : REFERENCE TO ARRAY[0..XtsCoreParameters.MAX_NUMBER_LOCAL_LOG - 1] OF I_XtsLogCommand
GET
DetailedCommands REF= _Entries;
END_GET
END_PROPERTY

//FB_Init is always available implicitly and it is used primarily for initialization.
//The return value is not evaluated. For a specific influence, you can also declare the
//methods explicitly and provide additional code there with the standard initialization
//code. You can evaluate the return value.
METHOD FB_Init: BOOL
VAR_INPUT
    bInitRetains: BOOL; // TRUE: the retain variables are initialized (reset warm / reset cold)
    bInCopyCode: BOOL;  // TRUE: the instance will be copied to the copy code afterward (online change)   
END_VAR
VAR
	i : UDINT;
END_VAR
FOR i:= 0 TO XtsCoreParameters.MAX_NUMBER_LOCAL_LOG - 1 DO
	_Entries[i] := _LogEntries[i];
END_FOR
END_METHOD

METHOD LogMessage
VAR_INPUT
	Key		  : T_MaxString;
	Value	  : T_MaxString;
	SourceId  : UDINT := 0;
	TimeStamp : ULINT := 0;
	MessageId : UDINT := 1;
	Severity  : USINT := 1;
END_VAR

VAR_INST
	LogSource  : TraceSourceInfo;
	LogMessage : TraceMessageInfo;
END_VAR
LogSource.SourceName := Key;
LogSource.SourceId	 := SourceId;
LogSource.TimeStamp	 := TimeStamp;
LogMessage.Message	 := Value;
LogMessage.MessageId := MessageId;
LogMessage.Severity	 := Severity;
THIS^.LogMessageInstance(LogSource, LogMessage);
END_METHOD

METHOD LogMessageInstance
VAR_INPUT
	SourceInfo	: I_TraceSourceInfo;
	MessageInfo : I_TraceMessageInfo;
	Arguments	: I_TraceArgument := 0;
END_VAR

VAR
	SysTime	 : T_FILETIME64;
	Severity : T_MaxString;
END_VAR
MEMMOVE(ADR(_SimpleLog[1]), ADR(_SimpleLog[0]), SIZEOF(_SimpleLog[0]) * (XtsCoreParameters.MAX_NUMBER_LOCAL_LOG - 1));
MEMMOVE(ADR(_LogEntries[1]), ADR(_LogEntries[0]), SIZEOF(_LogEntries[0]) * (XtsCoreParameters.MAX_NUMBER_LOCAL_LOG - 1));
_LogEntries[0].SourceId	  := SourceInfo.SourceId;
_LogEntries[0].SourceName := SourceInfo.SourceName;
IF SourceInfo.TimeStamp = 0 THEN
	SysTime					 := F_GetSystemTime();
	_LogEntries[0].Timestamp := SysTime;
ELSE
	_LogEntries[0].TimeStamp := SourceInfo.TimeStamp;
END_IF

_LogEntries[0].Message	 := MessageInfo.Message;
_LogEntries[0].MessageId := MessageInfo.MessageId;
_LogEntries[0].Severity	 := MessageInfo.Severity;
_LogEntries[0].Arguments := Arguments;
_SimpleLog[0]			 := CONCAT(SYSTEMTIME_TO_STRING(FILETIME64_TO_SYSTEMTIME(_LogEntries[0].TimeStamp)),
								   CONCAT(' ', CONCAT(GetSeverityString(MessageInfo.Severity), CONCAT(_LogEntries[0].SourceName, CONCAT(': ', _LogEntries[0].Message)))));

IF Arguments <> 0 THEN
	_SimpleLog[0] := CONCAT(_SimpleLog[0], Arguments.ToString());
END_IF
END_METHOD

END_FUNCTION_BLOCK

// Logging/Interfaces/I_XtsLocalLogger
INTERFACE I_XtsLocalLogger EXTENDS I_XtsLocalLog, I_XtsLogger

END_INTERFACE

// Logging/XtsLogCommand
{attribute 'hide_all_locals'}
FUNCTION_BLOCK XtsLogCommand IMPLEMENTS I_XtsLogCommand
VAR
	_MessageInfo : TraceMessageInfo;
	_SourceInfo	 : TraceSourceInfo;
	_Arguments	 : I_TraceArgument;
END_VAR

{attribute 'monitoring' := 'call'}
PROPERTY Arguments : I_TraceArgument
GET
Arguments := _Arguments;
END_GET
SET
_Arguments := Arguments;
END_SET
END_PROPERTY

{attribute 'monitoring':='call'}
PROPERTY Message : T_MaxString
GET
Message := _MessageInfo.Message;
END_GET
SET
_MessageInfo.Message := Message;
END_SET
END_PROPERTY

{attribute 'monitoring':='call'}
PROPERTY MessageId : UDINT
GET
MessageId := _MessageInfo.MessageId;
END_GET
SET
_MessageInfo.MessageId := MessageId;
END_SET
END_PROPERTY

{attribute 'monitoring':='call'}
PROPERTY Severity : USINT
GET
Severity := _MessageInfo.Severity;
END_GET
SET
_MessageInfo.Severity := Severity;
END_SET
END_PROPERTY

{attribute 'monitoring':='call'}
PROPERTY SourceId : UDINT
GET
SourceId := _SourceInfo.SourceId;
END_GET
SET
_SourceInfo.SourceId := SourceId;
END_SET
END_PROPERTY

{attribute 'monitoring':='call'}
PROPERTY SourceName : T_MaxString
GET
SourceName := _SourceInfo.SourceName;
END_GET
SET
_SourceInfo.SourceName := SourceName;
END_SET
END_PROPERTY

{attribute 'monitoring':='call'}
PROPERTY TimeStamp : ULINT
GET
TimeStamp := _SourceInfo.TimeStamp;
END_GET
SET
_SourceInfo.TimeStamp := TimeStamp;
END_SET
END_PROPERTY

END_FUNCTION_BLOCK

// _Internal/NullObjects/GetSeverityString
FUNCTION GetSeverityString : T_MaxString
VAR_INPUT
	Severity : USINT;
END_VAR
VAR
END_VAR

CASE Severity OF
	0:
		GetSeverityString := 'Verbose: ';

	1:
		GetSeverityString := 'Info: ';

	2:
		GetSeverityString := 'Warning: ';

	3:
		GetSeverityString := 'Error: ';

	4:
		GetSeverityString := 'Critical Error: ';

ELSE
	GetSeverityString := CONCAT('Severity: ', TO_STRING(Severity));
END_CASE

END_FUNCTION

// Logging/XtsTracePublisher
FUNCTION_BLOCK XtsTracePublisher IMPLEMENTS I_XtsTracePublisher
VAR
	{attribute 'hide'}
	_Subscribers : Collection;
END_VAR

METHOD LogMessage
VAR_INPUT
	Key		  : T_MaxString;
	Value	  : T_MaxString;
	SourceId  : UDINT := 0;
	TimeStamp : ULINT := 0;
	MessageId : UDINT := 1;
	Severity  : USINT := 1;
END_VAR

VAR
	Logger : I_TraceLogger;
END_VAR
_Subscribers.ResetIterator();
WHILE _Subscribers.MoveToNext DO
	__QUERYINTERFACE(_Subscribers.Current, Logger);
	IF Logger <> 0 THEN
		Logger.LogMessage(Key,
						  Value,
						  SourceId,
						  TimeStamp,
						  MessageId,
						  Severity);
	END_IF
END_WHILE
END_METHOD

METHOD LogMessageInstance
VAR_INPUT
	SourceInfo	: I_TraceSourceInfo;
	MessageInfo : I_TraceMessageInfo;
	Arguments	: I_TraceArgument := 0;
END_VAR

VAR
	Logger : I_TraceInstanceLogger;
END_VAR
_Subscribers.ResetIterator();
WHILE _Subscribers.MoveToNext DO
	__QUERYINTERFACE(_Subscribers.Current, Logger);
	IF Logger <> 0 THEN
		Logger.LogMessageInstance(SourceInfo, MessageInfo, Arguments);
	END_IF
END_WHILE
END_METHOD

METHOD Subscribe
VAR_INPUT
	Logger : I_XtsLogger;
END_VAR
_Subscribers.AddItem(Logger);
END_METHOD

METHOD Unsubscribe
VAR_INPUT
	Logger : I_XtsLogger;
END_VAR
_Subscribers.RemoveItem(Logger);
END_METHOD

END_FUNCTION_BLOCK

// _Internal/Mover/Properties/PositionableBehavior
{attribute 'no_explicit_call' := 'This FB is a CLASS and must be accessed using methods or properties'}
FUNCTION_BLOCK PositionableBehavior IMPLEMENTS I_AxisTrackPositionable, I_Cyclic
VAR
	_Axis			 : I_AxisRef;
	_MoverUtility	 : I_TcIoXtsXpuMover;
	_Position		 : LREAL;
	_ActualPositions : ST_PositionInfo;
END_VAR

PROPERTY Axis : I_AxisRef
GET
Axis := _Axis;
END_GET
SET
VAR
	Mover : I_XtsMover;
END_VAR
_Axis := Axis;
__QUERYINTERFACE(Axis, Mover);
 _MoverUtility := Mover.MoverUtility;
END_SET
END_PROPERTY

METHOD CyclicLogic
IF _MoverUtility = 0 THEN
	_Position := _Axis.Axis.NcToPlc.ModuloSetPos;
	RETURN;
END_IF
_ActualPositions := _MoverUtility.GetPositionInfo();
IF _ActualPositions.nTrackObjectid <> 0 THEN
	//We're on a track
	_Position := _ActualPositions.fTrackPosition;
ELSE
	//We're not, provide the modulo set position as the current position
	_Position := _Axis.Axis.NcToPlc.ModuloSetPos;
END_IF
END_METHOD

//FB_Init is always available implicitly and it is used primarily for initialization.

//The return value is not evaluated. For a specific influence, you can also declare the

//methods explicitly and provide additional code there with the standard initialization

//code. You can evaluate the return value.
METHOD FB_Init : BOOL
VAR_INPUT
	bInitRetains : BOOL; // TRUE: the retain variables are initialized (reset warm / reset cold)
	bInCopyCode	 : BOOL; // TRUE: the instance will be copied to the copy code afterward (online change)
	Axis		 : I_AxisRef;
END_VAR
VAR
	Mover : I_XtsMover;
END_VAR
_Axis := Axis;
__QUERYINTERFACE(Axis, Mover);
 _MoverUtility := Mover.MoverUtility;
END_METHOD

PROPERTY MoverUtility : I_TcIoXtsXpuMover
SET
_MoverUtility := MoverUtility;
END_SET
END_PROPERTY

{attribute 'monitoring':='call'}
PROPERTY PartPosition : LREAL
GET
PartPosition := _ActualPositions.fPartPosition;
END_GET
END_PROPERTY

{attribute 'monitoring':='call'}
PROPERTY Position : LREAL
GET
Position := _Position;
END_GET
END_PROPERTY

{attribute 'monitoring':='call'}
PROPERTY TrackPosition : LREAL
GET
TrackPosition := _ActualPositions.fTrackPosition;
END_GET
END_PROPERTY

END_FUNCTION_BLOCK

// _Internal/Mover/Properties/I_AxisTrackPositionable
INTERFACE I_AxisTrackPositionable EXTENDS I_Base

PROPERTY Axis : I_AxisRef
GET
END_GET
SET
END_SET
END_PROPERTY

PROPERTY MoverUtility : I_TcIoXtsXpuMover
SET
END_SET
END_PROPERTY

{attribute 'monitoring':='call'}
PROPERTY PartPosition : LREAL
GET
END_GET
END_PROPERTY

{attribute 'monitoring':='call'}
PROPERTY Position : LREAL
GET
END_GET
END_PROPERTY

{attribute 'monitoring':='call'}
PROPERTY TrackPosition : LREAL
GET
END_GET
END_PROPERTY

END_INTERFACE

// _Internal/Mover/Status/XtsMoverStatus
{attribute 'no_explicit_call' := 'This FB is a CLASS and must be accessed using methods or properties'}
{attribute 'conditionalshow'}
FUNCTION_BLOCK XtsMoverStatus IMPLEMENTS I_XtsMoverStatus
VAR
	_Axis			   : I_AxisRef;
	_CurrentTrack	   : I_XtsTrack := NullObjects.XtsTrack;
	_CommandedPosition : LREAL;
	_CommandedStation  : I_XtsStation := NullObjects.Station;
	_IdentInGroup	   : UDINT;
	_MoverInGroup	   : BOOL;
	_InSync			   : BOOL;
END_VAR

{attribute 'monitoring':='call'}
PROPERTY ActualAcceleration : LREAL
GET
ActualAcceleration := _Axis.Axis.NcToPlc.ActAcc;
END_GET
END_PROPERTY

{attribute 'monitoring':='call'}
PROPERTY ActualVelocity : LREAL
GET
ActualVelocity := _Axis.Axis.NcToPlc.ActVelo;
END_GET
END_PROPERTY

{attribute 'monitoring':='call'}
PROPERTY AvoidingCollision : BOOL
GET
AvoidingCollision := _Axis.Axis.NcToPlc.StateDWord2.Flags.AvoidingCollision;
END_GET
END_PROPERTY

{attribute 'monitoring':='call'}
PROPERTY Axis : I_AxisRef
GET
Axis := _Axis;
END_GET
END_PROPERTY

{attribute 'monitoring' := 'call'}
PROPERTY CommandedPosition : LREAL
GET
CommandedPosition := _CommandedPosition;
END_GET
SET
_CommandedPosition := CommandedPosition;
END_SET
END_PROPERTY

{attribute 'monitoring':='call'}
PROPERTY CommandedStation : I_XtsStation
GET
CommandedStation := _CommandedStation;
END_GET
SET
_CommandedStation := CommandedStation;
END_SET
END_PROPERTY

{attribute 'monitoring':='call'}
PROPERTY CurrentTrack : I_XtsTrack
GET
CurrentTrack := _CurrentTrack;
END_GET
SET
_CurrentTrack := CurrentTrack;
END_SET
END_PROPERTY

//FB_Init is always available implicitly and it is used primarily for initialization.
//The return value is not evaluated. For a specific influence, you can also declare the
//methods explicitly and provide additional code there with the standard initialization
//code. You can evaluate the return value.
METHOD FB_Init: BOOL
VAR_INPUT
    bInitRetains: BOOL; // TRUE: the retain variables are initialized (reset warm / reset cold)
    bInCopyCode: BOOL;  // TRUE: the instance will be copied to the copy code afterward (online change)   
	Axis : I_AxisRef;
END_VAR
_Axis := Axis;
END_METHOD

{attribute 'monitoring':='call'}
PROPERTY IdentInGroup : UDINT
GET
IdentInGroup := _IdentInGroup;
END_GET
SET
_IdentInGroup := IdentInGroup;
END_SET
END_PROPERTY

{attribute 'monitoring' := 'call'}
PROPERTY InSync : BOOL
GET
InSync := _InSync;
END_GET
SET
_InSync := InSync;
END_SET
END_PROPERTY

{attribute 'monitoring':='call'}
PROPERTY MoverInGroup : BOOL
GET
MoverInGroup := _IdentInGroup <> 0;
END_GET
END_PROPERTY

{attribute 'monitoring':='call'}
PROPERTY SetAcceleration : LREAL
GET
SetAcceleration := _Axis.Axis.NcToPlc.SetAcc;
END_GET
END_PROPERTY

{attribute 'monitoring':='call'}
PROPERTY SetVelocity : LREAL
GET
SetVelocity := _Axis.Axis.NcToPlc.SetVelo;
END_GET
END_PROPERTY

END_FUNCTION_BLOCK

// _Internal/XtsSystem/Tasks/InitializeXtsTask
{attribute 'no_explicit_call' := 'This FB is a CLASS and must be accessed using methods or properties'}
FUNCTION_BLOCK InitializeXtsTask EXTENDS XtsTaskResult IMPLEMENTS I_XtsInitializeTask
VAR
	_XpuId				  : I_XtsXpuId;
	_XpuTcIoIndex		  : UINT;
	_XtsSystem			  : I_XtsSystem;
	_XtsUtilityProperties : I_ContainXtsSystemProperties;
	_XtsUtility			  : I_ContainXtsUtility;
	_State				  : UDINT;
	_SubState			  : UDINT;
	i					  : UDINT;
	MoverCommander		  : XtsMoverCommander;
	_Initialized		  : BOOL;

	//
	XtsEnvironmentFB			: FB_TcIoXtsEnvironment;
	_XtsEnvironment				: I_TcIoXtsEnvironment := XtsEnvironmentFB;
	XtsEnvironmentConfiguration : ST_XtsEnvironmentConfiguration;
	_Xpu						: I_TcIoXtsProcessingUnit;
	_InfoServer					: I_TcIoXtsInfoServer;
	_InfoServerOTCID			: UDINT;
	_TrackCollection			: I_ContainXtsTracks;
	_PartCollection				: I_ContainXtsParts;

	//
	_MoverDetectTask   : I_XtsTask;
	_MoverRedetectTask : I_XtsTask;
	_MoverIDTask	   : I_XtsTask;
END_VAR

METHOD Initialize
VAR
	LogSource  : TraceSourceInfo;
	LogMessage : TraceMessageInfo;
END_VAR
CASE _State OF
	0:
		IF _Initialized THEN
			RETURN;
		END_IF

		_Busy										   := TRUE;
		_Error										   := FALSE;
		_ErrorId									   := 0;
		XtsEnvironmentConfiguration.bEnableInitCaGroup := TRUE;
		_XtsEnvironment.P_XtsEnvironmentConfiguration  REF= XtsEnvironmentConfiguration;
		_State										   := 10;
		LogSource.SourceName						   := 'InitializeXtsTask';
		LogMessage.Message							   := 'Iinitialization started.';
		LogMessage.MessageId						   := E_XtsLogMessage.SystemInitializationStarted;
		LogMessage.Severity							   := 1;
		_Logger.LogMessageInstance(LogSource, LogMessage);

	10:
		IF _XtsEnvironment.Init(TRUE) THEN
			_XtsEnvironment.Init(FALSE);
			_State := 20;
		END_IF

	20:
		IF NOT _XtsEnvironment.P_IsInitialized THEN
			_Error				 := TRUE;
			_ErrorId			 := E_XtsLogMessage.SystemError;
			LogMessage.Message	 := 'Environment Not Initialized';
			LogMessage.MessageId := E_XtsLogMessage.SystemError;
			LogMessage.Severity	 := 3;
			_Logger.LogMessageInstance(LogSource, LogMessage);
			Trace.LogMessage(Key	   := LogSource.SourceName,
							 Value	   := LogMessage.Message,
							 MessageId := LogMessage.MessageId,
							 Severity  := LogMessage.Severity);

			_State := 65535;
		ELSE
			_XtsSystem.Environment := _XtsEnvironment;
			IF _XtsEnvironment.GetXpuCount(TRUE) THEN
				_XtsEnvironment.GetXpuCount(FALSE);
				i	   := 1;
				_State := 21;
			END_IF
		END_IF

	21:
	
		IF _XtsEnvironment.XpuTcIo(UDINT_TO_UINT(i)).P_ObjectName = _XtsSystem.Name THEN
			_XtsSystem.Utility := _Xpu := _XtsEnvironment.XpuTcIo(UDINT_TO_UINT(i));
			_XpuTcIoIndex			   := UDINT_TO_UINT(i);
			_State					   := 30;
		ELSE
			i := i + 1;
			IF i > _XtsEnvironment.P_XpuCountUint THEN
				LogMessage.Message	 := 'XPU Name not found! Ensure XtsSystem declaration name matches TcCom object name';
				LogMessage.MessageId := E_XtsLogMessage.SystemInitializationXpuNameNotFound;
				LogMessage.Severity	 := 3;
				_Logger.LogMessageInstance(LogSource, LogMessage);
				Trace.LogMessage(Key	   := LogSource.SourceName,
								 Value	   := LogMessage.Message,
								 MessageId := LogMessage.MessageId,
								 Severity  := LogMessage.Severity);

				_Error	 := TRUE;
				_ErrorId := E_XtsLogMessage.SystemInitializationXpuNameNotFound;
				_State	 := 65535;
			END_IF
		END_IF

	30:
		IF MoverSetup() THEN
			LogSource.SourceName := 'InitializeXtsTask';
			LogMessage.Message	 := 'Mover Initialization Finished.';
			LogMessage.MessageId := E_XtsLogMessage.SystemMoverInitializationFinished;
			LogMessage.Severity	 := 0;
			_Logger.LogMessageInstance(LogSource, LogMessage);
			_State := 31;
		END_IF

	31:
		IF InfoServerSetup() THEN
			LogSource.SourceName := 'InitializeXtsTask';
			LogMessage.Message	 := 'Infoserver Initialization Finished.';
			LogMessage.MessageId := E_XtsLogMessage.SystemVerbose;
			LogMessage.Severity	 := 0;
			_Logger.LogMessageInstance(LogSource, LogMessage);
			_State := 40;
		END_IF

	40:
		IF TrackSetup() THEN
			_State := 41;
		END_IF

	41:
		//Make sure AxesGroupRef is linked
		IF _XtsSystem.AxesGroupRef.NcToPlc.CA.Common.GroupOID = 0 THEN
			LogSource.SourceName := 'InitializeXtsTask';
			LogMessage.Message	 := 'XtsSystem AxesGroupRef is not linked!';
			LogMessage.MessageId := E_XtsLogMessage.SystemInitializationAxesGroupNotLinked;
			LogMessage.Severity	 := 3;
			Trace.LogMessage(Key	   := LogSource.SourceName,
							 Value	   := LogMessage.Message,
							 MessageId := LogMessage.MessageId,
							 Severity  := LogMessage.Severity);

			_Logger.LogMessageInstance(LogSource, LogMessage);
			_ErrorId := E_XtsLogMessage.SystemInitializationAxesGroupNotLinked;
			_Error	 := TRUE;
			_State	 := 65535;
		ELSE
			_State := 42;
		END_IF

	42:
		IF _XtsSystem.Environment.GetCaGroupOids(TRUE) THEN
			_XtsSystem.Environment.GetCaGroupCount(FALSE);
			i	   := 1;
			_State := 43;
		END_IF

